Fanuc TP program (LS listing): JOB_VAR_OD_GRIP.LS

/PROG  JOB_VAR_OD_GRIP
/ATTR
OWNER		= MNEDITOR;
COMMENT		= "";
PROG_SIZE	= 93425;
CREATE		= DATE 19-07-31  TIME 17:01:20;
MODIFIED	= DATE 26-06-08  TIME 14:37:38;
FILE_NAME	= JOB_VARI;
VERSION		= 0;
LINE_COUNT = 3201;
MEMORY_SIZE	= 94489;
PROTECT		= READ_WRITE;
TCD:  STACK_SIZE	= 0,
      TASK_PRIORITY	= 50,
      TIME_SLICE	= 0,
      BUSY_LAMP_OFF	= 0,
      ABORT_REQUEST	= 0,
      PAUSE_REQUEST	= 0;
DEFAULT_GROUP	= 1,*,*,*,*;
CONTROL_CODE	= 00000000 00000000;
/APPL

AUTO_SINGULARITY_HEADER;
  ENABLE_SINGULARITY_AVOIDANCE   : TRUE;
/MN
   1:  !R[70] is the item number ;
   2:  !R[71] if using previous data ;
   3:  R[196]=AR[1]    ;
   4:  R[197]=AR[2]    ;
   5:  !------------------------- ;
   6:  !Item Select = 102680550 ;
   7:  SELECT R[70]=550,JMP LBL[550] ;
   8:  !Item Select = 102680552 ;
   9:         =552,JMP LBL[552] ;
  10:  !Item Select = MEC0253 ;
  11:         =253,JMP LBL[253] ;
  12:  !Item Select = 102680551 ;
  13:         =551,JMP LBL[551] ;
  14:  !Item Select = 1090747 ;
  15:         =747,JMP LBL[747] ;
  16:  !Item Select = 102772049 ;
  17:         =2049,JMP LBL[2049] ;
  18:  !Item Select = 102712760 ;
  19:         =2760,JMP LBL[2760] ;
  20:  !Item Select = 102740005 ;
  21:         =4005,JMP LBL[4005] ;
  22:  !Item Select = 103044540 ;
  23:         =4540,JMP LBL[4540] ;
  24:  !Item Select = 102824679 ;
  25:         =4679,JMP LBL[4679] ;
  26:  !Item Select = 103095029 ;
  27:         =5029,JMP LBL[5029] ;
  28:  !Item Select = 1025649 ;
  29:         =5649,JMP LBL[5649] ;
  30:  !Item Select = 103365943 ;
  31:         =5943,JMP LBL[5943] ;
  32:  !Item Select = 102906372 ;
  33:         =6372,JMP LBL[6372] ;
  34:  !Item Select = 102666549 ;
  35:         =6549,JMP LBL[6549] ;
  36:  !Item Select = 1026588 ;
  37:         =6588,JMP LBL[6588] ;
  38:  !Item Select = 1026617 ;
  39:         =6617,JMP LBL[6617] ;
  40:  !Item Select = 102606754 ;
  41:         =6754,JMP LBL[6754] ;
  42:  !Item Select = 102606755 ;
  43:         =6755,JMP LBL[6755] ;
  44:  !Item Select = 102757062 ;
  45:         =7062,JMP LBL[7062] ;
  46:  !Item Select = 102577436 ;
  47:         =7436,JMP LBL[7436] ;
  48:  !Item Select = 1017688 ;
  49:         =7688,JMP LBL[7688] ;
  50:  !Item Select = 207757 ;
  51:         =7757,JMP LBL[7757] ;
  52:  !Item Select = 198034 ;
  53:         =8034,JMP LBL[8034] ;
  54:  !Item Select = 102678902 ;
  55:         =8902,JMP LBL[8902] ;
  56:  !Item Select = 102709487 ;
  57:         =9487,JMP LBL[9487] ;
  58:  !Item Select = 100009654 ;
  59:         =9654,JMP LBL[9654] ;
  60:  !Item Select = 102779700 ;
  61:         =9700,JMP LBL[9700] ;
  62:  !Item Select = 102649814 ;
  63:         =9814,JMP LBL[9814] ;

  64:  !Item Select = 111199990 ;
  65:         =9990,JMP LBL[9990] ;


  66:  !No conditions are met, jump ;
  67:  !to the very end of the program ;
  68:         ELSE,JMP LBL[9999] ;
  69:   ;
  70:  LBL[253] ;
  71:  !--------------------------- ;
  72:  !HANDLE PULL ;
  73:  !Item MEC0253, Rev 01-000 ;
  74:  !Last Modified: 2025-07-25 ;
  75:  !Modified by: AARON ;
  76:  !0.35 IN Height ;
  77:  !0.09 IN ID, 0.25 IN OD ;
  78:  !OD Jaw #1005 ;
  79:  !------------------------- ;
  80:  IF (R[70]=253) THEN ;
  81:   ;
  82:  !Define Parameters for INF/OTF ;
  83:  !R[105]=AR[1]=100, 2By3 Sheet ;
  84:  !R[105]=AR[1]=200, 3By4 Sheet ;
  85:  !R[105]=AR[1]=300, 5By7 Sheet ;
  86:  CALL JOB_VAR_SETUP(200) ;
  87:   ;
  88:  !------------------------- ;
  89:  !Define Parameters for Job ;
  90:  R[1]=0    ;
  91:  R[67]=20    ;
  92:  R[2]=0    ;
  93:  R[3]=1    ;
  94:  R[139]=12    ;
  95:  R[4]=0    ;
  96:  R[85]=64    ;
  97:  R[86]=5    ;
  98:  R[87]=150    ;
  99:  R[95]=100    ;
 100:  R[110]=2026    ;
 101:  !CNC W-AXIS OFFSET ;
 102:  R[111]=((-16.06)) ;
 103:  !X-Compliance Push Bypass ;
 104:  F[6:OFF]=(OFF) ;
 105:  !--------------------------- ;
 106:  !R[100] "GRIPPER_ID" 3 values ;
 107:  !If =100, ID Grippers Installed ;
 108:  !If =200, OD Grippers Installed ;
 109:  !If =300, OD 45 Degree Grippers ;
 110:  R[100]=200    ;
 111:  !--------------------------- ;
 112:   ;
 113:  !If using previous setup data ;
 114:  IF (R[71]=253) THEN ;
 115:   ;
 116:  !--------------------------- ;
 117:  R[190]=20.5    ;
 118:  R[191]=15.798    ;
 119:  R[192]=(-36)    ;
 120:  R[193]=(-440)    ;
 121:  !--------------------------- ;
 122:   ;
 123:   ;
 124:  CALL CREATE_REG(R[190],R[191],R[192],R[193]) ;
 125:   ;
 126:  ENDIF ;
 127:   ;
 128:  !If new loading or offloading pos ;
 129:  !SET R[104] "IMPORT_LOADPOS" ;
 130:  !SET R[104]=1000, Otherwise NO ;
 131:  R[104]=1000    ;
 132:  IF (R[104]=1000) THEN ;
 133:  !R[260]=43, Preload Pos1 ;
 134:  !R[270]=44, Preload PosFinal ;
 135:  !R[300]=53, Offload PosFinal ;
 136:  !PR[43] Pre-Loading Pos1 ;
 137:  CALL CREATE_PR(43,167.761,(-61.029),337.113,(-171.936),88.039,(-174.046)) ;
 138:  !PR[44] Final Loading Position ;
 139:  CALL CREATE_PR(44,168.578,(-60.735),361.702,(-171.929),88.036,(-174.03)) ;
 140:  !PR[53] Pre Unloading Position ;
 141:  CALL CREATE_PR(53,(-127.197),94.302,111.215,163.187,(-88.443),(-162.218)) ;
 142:  !PR[54] Final Unloading Position ;
 143:  CALL CREATE_PR(54,(-125.519),94.106,49.029,163.508,(-88.445),(-162.507)) ;
 144:  ENDIF ;
 145:   ;
 146:  !---------------------------- ;
 147:  !SR[2] = "JOB_VAR_OD_GRIP" ;
 148:  !JOB_VAR_COMMON(R[103])'s value ;
 149:  !---------------------------- ;
 150:  !2By3 SR[2] INF, Max 18(Straight) ;
 151:  !R[103]=200 ;
 152:  !2By3 INF 45 Degree Diagonal Shif ;
 153:  !R[103]=210 ;
 154:  !---------------------------- ;
 155:  !3By4 SR[2] INF, Max 36(Straight) ;
 156:  !R[103]=250 ;
 157:  !3By4 INF 45 Degree Diagonal Shif ;
 158:  !R[103]=260 ;
 159:  !---------------------------- ;
 160:  !R[103] "JOB_PROFILE" Selection ;
 161:  R[103]=250    ;
 162:  CALL JOB_VAR_COMMON(R[103]) ;
 163:   ;
 164:  ENDIF ;
 165:   ;
 166:  JMP LBL[9999] ;
 167:   ;
 168:  !Job MEC0253 Logic Ends ;
 169:  !--------------------------- ;
 170:   ;
 171:  LBL[550] ;
 172:  !--------------------------- ;
 173:  !Thimble Upper ;
 174:  !Item 102680550 , Rev A ;
 175:  !Last Modified: 2024-06-24 ;
 176:  !Modified by: SH ;
 177:  !1.06 IN Height ;
 178:  !3.3 IN ID, 4.49 IN OD ;
 179:  !OD Jaw # 2003 ;
 180:  !--------------------------- ;
 181:  IF (R[70]=550) THEN ;
 182:  !Define Parameters for INF/OTF ;
 183:  !R[105]=AR[1]=100, 2By3 Sheet ;
 184:  !R[105]=AR[1]=200, 3By4 Sheet ;
 185:  !R[105]=AR[1]=300, 5By7 Sheet ;
 186:  CALL JOB_VAR_SETUP(100) ;
 187:   ;
 188:  !--------------------------- ;
 189:  !Define Parameters for Job ;
 190:  R[1]=1    ;
 191:  R[67]=20    ;
 192:  R[2]=0    ;
 193:  R[139]=12    ;
 194:  !R[85] "INF_JAW_OFFSET"(Hgt) ;
 195:  R[85]=92.05    ;
 196:  !R[86] "INF_PICK_OFFSET" 50mm/sec ;
 197:  R[86]=5    ;
 198:  !R[87] "MAIN_LOAD_OFFSET" (PRELOA ;
 199:  R[87]=100    ;
 200:  !R[100] "GRIPPER_ID" 3 values ;
 201:  !If =100, ID Grippers Installed ;
 202:  !If =200, OD Grippers Installed ;
 203:  !If =300, OD 45 Degree Grippers ;
 204:  R[100]=200    ;
 205:  !--------------------------- ;
 206:   ;
 207:  !If using previous setup data ;
 208:  IF (R[71]=550) THEN ;
 209:   ;
 210:  !--------------------------- ;
 211:  !1st: Height of Raw piece ;
 212:  R[190]=32.2    ;
 213:  !2nd: Height of Finish piece ;
 214:  R[191]=27    ;
 215:  !3rd: Infeed Height Offset ;
 216:  R[192]=(-240)    ;
 217:  !4th: Outfeed Height Offset ;
 218:  R[193]=(-285)    ;
 219:  !--------------------------- ;
 220:   ;
 221:  CALL CREATE_REG(R[190],R[191],R[192],R[193]) ;
 222:   ;
 223:  ENDIF ;
 224:   ;
 225:  !If new loading or offloading pos ;
 226:  !SET R[104] "IMPORT_LOADPOS" ;
 227:  !SET R[104]=1000, Otherwise NO ;
 228:  R[104]=1000    ;
 229:  IF (R[104]=1000) THEN ;
 230:  !R[260]=43, Preload Pos1 ;
 231:  !R[270]=44, Preload PosFinal ;
 232:  !R[300]=53, Offload PosFinal ;
 233:  !PR[43] Pre-Loading Pos1 ;
 234:  CALL CREATE_PR(43,167.274,(-59.505),319.711,168.214,88.493,166.138) ;
 235:  !PR[44] Final Loading Position ;
 236:  CALL CREATE_PR(44,167.813,(-59.797),340.237,168.005,88.489,165.921) ;
 237:  !PR[53] Pre Unloading Position ;
 238:  CALL CREATE_PR(53,(-127.387),93.873,91.227,168.522,(-88.33),(-169.447)) ;
 239:  !PR[54] Final Unloading Position ;
 240:  CALL CREATE_PR(54,(-126.716),94.154,67.135,168.491,(-88.33),(-169.421)) ;
 241:  !PR[56] assitant Unloading preses ;
 242:  CALL CREATE_PR(56,(-131.536),105.713,233.177,173.746,(-88.233),(-175.647)) ;
 243:  !PR[57] assitant Unloading preses ;
 244:  CALL CREATE_PR(57,(-133.703),92.431,364.782,167.802,(-88.383),(-166.755)) ;
 245:  !PR[58] assitant Unloading preses ;
 246:  CALL CREATE_PR(58,(-133.703),92.431,364.782,167.804,(-88.383),(-166.755)) ;
 247:  ENDIF ;
 248:   ;
 249:  !---------------------------- ;
 250:  !SR[2] = "JOB_VAR_OD_GRIP" ;
 251:  !JOB_VAR_COMMON(R[103])'s value ;
 252:  !---------------------------- ;
 253:  !2By3 SR[2] INF, Max 18(Straight) ;
 254:  !R[103]=200 ;
 255:  !2By3 INF 45 Degree Diagonal Shif ;
 256:  !R[103]=210 ;
 257:  !---------------------------- ;
 258:  !3By4 SR[2] INF, Max 36(Straight) ;
 259:  !R[103]=250 ;
 260:  !3By4 INF 45 Degree Diagonal Shif ;
 261:  !R[103]=260 ;
 262:  !---------------------------- ;
 263:  !R[103] "JOB_PROFILE" Selection ;
 264:  R[103]=200    ;
 265:  CALL JOB_VAR_COMMON(R[103]) ;
 266:   ;
 267:  ENDIF ;
 268:   ;
 269:  JMP LBL[9999] ;
 270:   ;
 271:  !Job 102680550 Logic Ends ;
 272:  !--------------------------- ;
 273:   ;
 274:  LBL[551] ;
 275:  !--------------------------- ;
 276:  !Thimble Lower ;
 277:  !Item 102680551 , Rev A ;
 278:  !Last Modified: 2026-05-20 ;
 279:  !Modified by: Aaron ;
 280:  !1.38 IN Height ;
 281:  !3.372 IN ID, 4.49 IN OD ;
 282:  !OD Jaw # 2002 ;
 283:  !--------------------------- ;
 284:  IF (R[70]=551) THEN ;
 285:  !Define Parameters for INF/OTF ;
 286:  !R[105]=AR[1]=100, 2By3 Sheet ;
 287:  !R[105]=AR[1]=200, 3By4 Sheet ;
 288:  !R[105]=AR[1]=300, 5By7 Sheet ;
 289:  CALL JOB_VAR_SETUP(100) ;
 290:   ;
 291:  !--------------------------- ;
 292:  !Define Parameters for Job ;
 293:  R[1]=1    ;
 294:  R[67]=20    ;
 295:  R[2]=1    ;
 296:  R[139]=12    ;
 297:  !R[85] "INF_JAW_OFFSET"(Hgt) ;
 298:  R[85]=92.05    ;
 299:  !R[86] "INF_PICK_OFFSET" 50mm/sec ;
 300:  R[86]=10    ;
 301:  !R[87] "MAIN_LOAD_OFFSET" (PRELOA ;
 302:  R[87]=100    ;
 303:  !R[100] "GRIPPER_ID" 3 values ;
 304:  !If =100, ID Grippers Installed ;
 305:  !If =200, OD Grippers Installed ;
 306:  !If =300, OD 45 Degree Grippers ;
 307:  R[100]=200    ;
 308:  !--------------------------- ;
 309:   ;
 310:  !If using previous setup data ;
 311:  IF (R[71]=551) THEN ;
 312:   ;
 313:  !--------------------------- ;
 314:  !1st: Height of Raw piece ;
 315:  R[190]=41.5    ;
 316:  !2nd: Height of Finish piece ;
 317:  R[191]=35.05    ;
 318:  !3rd: Infeed Height Offset ;
 319:  R[192]=(-250)    ;
 320:  !4th: Outfeed Height Offset ;
 321:  R[193]=(-280)    ;
 322:  !--------------------------- ;
 323:   ;
 324:  CALL CREATE_REG(R[190],R[191],R[192],R[193]) ;
 325:   ;
 326:  ENDIF ;
 327:   ;
 328:  !If new loading or offloading pos ;
 329:  !SET R[104] "IMPORT_LOADPOS" ;
 330:  !SET R[104]=1000, Otherwise NO ;
 331:  R[104]=1000    ;
 332:  IF (R[104]=1000) THEN ;
 333:  !R[260]=43, Preload Pos1 ;
 334:  !R[270]=44, Preload PosFinal ;
 335:  !R[300]=53, Offload PosFinal ;
 336:  !PR[43] Pre-Loading Pos1 ;
 337:  CALL CREATE_PR(43,166.588,(-60.843),303.6,142.233,88.871,140.108) ;
 338:  !PR[44] Final Loading Position ;
 339:  CALL CREATE_PR(44,167.032,(-61.379),332.527,142.158,88.868,140.022) ;
 340:  !PR[53] Pre Unloading Position ;
 341:  CALL CREATE_PR(53,(-128.024),95.156,112.32,168.042,(-88.32),(-169.031)) ;
 342:  !PR[54] Final Unloading Position ;
 343:  CALL CREATE_PR(54,(-126.891),94.757,73.15,168.209,(-88.331),(-169.169)) ;
 344:  !PR[56] assitant Unloading preses ;
 345:  CALL CREATE_PR(56,(-131.536),105.713,233.177,173.746,(-88.233),(-175.647)) ;
 346:  !PR[57] assitant Unloading preses ;
 347:  CALL CREATE_PR(57,(-133.703),92.431,364.782,167.802,(-88.383),(-166.755)) ;
 348:  !PR[58] assitant Unloading preses ;
 349:  CALL CREATE_PR(58,(-133.703),92.431,364.782,167.804,(-88.383),(-166.755)) ;
 350:  ENDIF ;
 351:   ;
 352:  !---------------------------- ;
 353:  !SR[2] = "JOB_VAR_OD_GRIP" ;
 354:  !JOB_VAR_COMMON(R[103])'s value ;
 355:  !---------------------------- ;
 356:  !2By3 SR[2] INF, Max 18(Straight) ;
 357:  !R[103]=200 ;
 358:  !2By3 INF 45 Degree Diagonal Shif ;
 359:  !R[103]=210 ;
 360:  !---------------------------- ;
 361:  !3By4 SR[2] INF, Max 36(Straight) ;
 362:  !R[103]=250 ;
 363:  !3By4 INF 45 Degree Diagonal Shif ;
 364:  !R[103]=260 ;
 365:  !---------------------------- ;
 366:  !R[103] "JOB_PROFILE" Selection ;
 367:  R[103]=200    ;
 368:  CALL JOB_VAR_COMMON(R[103]) ;
 369:   ;
 370:  ENDIF ;
 371:   ;
 372:  JMP LBL[9999] ;
 373:   ;
 374:  !Job 102680551 Logic Ends ;
 375:  !--------------------------- ;
 376:   ;
 377:  LBL[552] ;
 378:  !--------------------------- ;
 379:  !COLLAR ;
 380:  !Item 102680552 , Rev A ;
 381:  !Last Modified: 2024-06-25 ;
 382:  !Modified by: TSUU ;
 383:  !1.79 IN Height ;
 384:  !3.110 IN ID, 3.56 IN OD ;
 385:  !OD Jaw # 2002 ;
 386:  !--------------------------- ;
 387:  IF (R[70]=552) THEN ;
 388:  !Define Parameters for INF/OTF ;
 389:  !R[105]=AR[1]=100, 2By3 Sheet ;
 390:  !R[105]=AR[1]=200, 3By4 Sheet ;
 391:  !R[105]=AR[1]=300, 5By7 Sheet ;
 392:  CALL JOB_VAR_SETUP(100) ;
 393:   ;
 394:  !--------------------------- ;
 395:  !Define Parameters for Job ;
 396:  R[1]=1    ;
 397:  R[67]=20    ;
 398:  R[2]=1    ;
 399:  R[139]=12    ;
 400:  !R[85] "INF_JAW_OFFSET"(Hgt) ;
 401:  R[85]=200    ;
 402:  !R[86] "INF_PICK_OFFSET" 50mm/sec ;
 403:  R[86]=15    ;
 404:  !R[87] "MAIN_LOAD_OFFSET" (PRELOA ;
 405:  R[87]=100    ;
 406:  !R[100] "GRIPPER_ID" 3 values ;
 407:  !If =100, ID Grippers Installed ;
 408:  !If =200, OD Grippers Installed ;
 409:  !If =300, OD 45 Degree Grippers ;
 410:  R[100]=200    ;
 411:  !--------------------------- ;
 412:   ;
 413:  !If using previous setup data ;
 414:  IF (R[71]=552) THEN ;
 415:   ;
 416:  !--------------------------- ;
 417:  !1st: Height of Raw piece ;
 418:  R[190]=50.546    ;
 419:  !2nd: Height of Finish piece ;
 420:  R[191]=45.46    ;
 421:  !3rd: Infeed Height Offset ;
 422:  R[192]=(-250)    ;
 423:  !4th: Outfeed Height Offset ;
 424:  R[193]=(-250)    ;
 425:  !--------------------------- ;
 426:   ;
 427:  CALL CREATE_REG(R[190],R[191],R[192],R[193]) ;
 428:   ;
 429:  ENDIF ;
 430:   ;
 431:  !If new loading or offloading pos ;
 432:  !SET R[104] "IMPORT_LOADPOS" ;
 433:  !SET R[104]=1000, Otherwise NO ;
 434:  R[104]=1000    ;
 435:  IF (R[104]=1000) THEN ;
 436:  !R[260]=43, Preload Pos1 ;
 437:  !R[270]=44, Preload PosFinal ;
 438:  !R[300]=53, Offload PosFinal ;
 439:  !PR[43] Pre-Loading Pos1 ;
 440:  CALL CREATE_PR(43,167.759,(-61.04),294.256,160.46,89.14,158.531) ;
 441:  !PR[44] Final Loading Position ;
 442:  CALL CREATE_PR(44,168.25,(-61.377),329.133,160.345,89.147,158.399) ;
 443:  !PR[53] Pre Unloading Position ;
 444:  CALL CREATE_PR(53,(-129.89),93.66,171.06,156.59,(-88.74),(-166.46)) ;
 445:  !PR[54] Final Unloading Position ;
 446:  CALL CREATE_PR(54,(-129),93.98,128.255,156.535,(-88.747),(-166.399)) ;
 447:  !PR[56] assitant Unloading preses ;
 448:  CALL CREATE_PR(56,(-131.536),105.713,233.177,173.746,(-88.233),(-175.647)) ;
 449:  !PR[57] assitant Unloading preses ;
 450:  CALL CREATE_PR(57,(-133.703),92.431,364.782,167.802,(-88.383),(-166.755)) ;
 451:  !PR[58] assitant Unloading preses ;
 452:  CALL CREATE_PR(58,(-133.703),92.431,364.782,167.804,(-88.383),(-166.755)) ;
 453:  ENDIF ;
 454:   ;
 455:  !---------------------------- ;
 456:  !SR[2] = "JOB_VAR_OD_GRIP" ;
 457:  !JOB_VAR_COMMON(R[103])'s value ;
 458:  !---------------------------- ;
 459:  !2By3 SR[2] INF, Max 18(Straight) ;
 460:  !R[103]=200 ;
 461:  !2By3 INF 45 Degree Diagonal Shif ;
 462:  !R[103]=210 ;
 463:  !---------------------------- ;
 464:  !3By4 SR[2] INF, Max 36(Straight) ;
 465:  !R[103]=250 ;
 466:  !3By4 INF 45 Degree Diagonal Shif ;
 467:  !R[103]=260 ;
 468:  !---------------------------- ;
 469:  !R[103] "JOB_PROFILE" Selection ;
 470:  R[103]=200    ;
 471:  CALL JOB_VAR_COMMON(R[103]) ;
 472:   ;
 473:  ENDIF ;
 474:   ;
 475:  JMP LBL[9999] ;
 476:   ;
 477:  !Job 102680552 Logic Ends ;
 478:  !--------------------------- ;
 479:   ;
 480:  LBL[747] ;
 481:  !--------------------------- ;
 482:  !PORT-GROVE VENT, JUICEBOX ;
 483:  !Item 1090747, Rev A ;
 484:  !Last Modified: 2025-03-22 ;
 485:  !Modified by: ZAMAN ;
 486:  !0.622 IN Height ;
 487:  !1.202 IN ID, 3.00 IN OD ;
 488:  !OD Jaw #2009 ;
 489:  !------------------------- ;
 490:  IF (R[70]=747) THEN ;
 491:   ;
 492:  !Define Parameters for INF/OTF ;
 493:  !R[105]=AR[1]=100, 2By3 Sheet ;
 494:  !R[105]=AR[1]=200, 3By4 Sheet ;
 495:  !R[105]=AR[1]=300, 5By7 Sheet ;
 496:  CALL JOB_VAR_SETUP(200) ;
 497:   ;
 498:  !------------------------- ;
 499:  !Define Parameters for Job ;
 500:  R[1]=1    ;
 501:  R[67]=20    ;
 502:  R[2]=0    ;
 503:  R[139]=12    ;
 504:  R[3]=0    ;
 505:  R[4]=0    ;
 506:  R[85]=64    ;
 507:  R[86]=5    ;
 508:  R[87]=150    ;
 509:  R[95]=100    ;
 510:  R[110]=2026    ;
 511:  !CNC W-AXIS OFFSET ;
 512:  R[111]=((-16.06)) ;
 513:  !X-Compliance Push Bypass ;
 514:  F[6:OFF]=(OFF) ;
 515:  !--------------------------- ;
 516:  !R[100] "GRIPPER_ID" 3 values ;
 517:  !If =100, ID Grippers Installed ;
 518:  !If =200, OD Grippers Installed ;
 519:  !If =300, OD 45 Degree Grippers ;
 520:  R[100]=200    ;
 521:  !--------------------------- ;
 522:   ;
 523:  !If using previous setup data ;
 524:  IF (R[71]=747) THEN ;
 525:   ;
 526:  !--------------------------- ;
 527:  R[190]=20.5    ;
 528:  R[191]=15.798    ;
 529:  R[192]=(-36)    ;
 530:  R[193]=(-498)    ;
 531:  !--------------------------- ;
 532:   ;
 533:   ;
 534:  CALL CREATE_REG(R[190],R[191],R[192],R[193]) ;
 535:   ;
 536:  ENDIF ;
 537:   ;
 538:  !If new loading or offloading pos ;
 539:  !SET R[104] "IMPORT_LOADPOS" ;
 540:  !SET R[104]=1000, Otherwise NO ;
 541:  R[104]=1000    ;
 542:  IF (R[104]=1000) THEN ;
 543:  !R[260]=43, Preload Pos1 ;
 544:  !R[270]=44, Preload PosFinal ;
 545:  !R[300]=53, Offload PosFinal ;
 546:  !PR[43] Pre-Loading Pos1 ;
 547:  CALL CREATE_PR(43,167.761,(-61.029),337.113,(-171.936),88.039,(-174.046)) ;
 548:  !PR[44] Final Loading Position ;
 549:  CALL CREATE_PR(44,168.578,(-60.735),361.702,(-171.929),88.036,(-174.03)) ;
 550:  !PR[53] Pre Unloading Position ;
 551:  CALL CREATE_PR(53,(-127.197),94.302,111.215,163.187,(-88.443),(-162.218)) ;
 552:  !PR[54] Final Unloading Position ;
 553:  CALL CREATE_PR(54,(-125.536),94.555,48.721,163.38,(-88.442),(-162.397)) ;
 554:  ENDIF ;
 555:   ;
 556:  !---------------------------- ;
 557:  !SR[2] = "JOB_VAR_OD_GRIP" ;
 558:  !JOB_VAR_COMMON(R[103])'s value ;
 559:  !---------------------------- ;
 560:  !2By3 SR[2] INF, Max 18(Straight) ;
 561:  !R[103]=200 ;
 562:  !2By3 INF 45 Degree Diagonal Shif ;
 563:  !R[103]=210 ;
 564:  !---------------------------- ;
 565:  !3By4 SR[2] INF, Max 36(Straight) ;
 566:  !R[103]=250 ;
 567:  !3By4 INF 45 Degree Diagonal Shif ;
 568:  !R[103]=260 ;
 569:  !---------------------------- ;
 570:  !R[103] "JOB_PROFILE" Selection ;
 571:  R[103]=250    ;
 572:  CALL JOB_VAR_COMMON(R[103]) ;
 573:   ;
 574:  ENDIF ;
 575:   ;
 576:  JMP LBL[9999] ;
 577:   ;
 578:  !Job 1090747 Logic Ends ;
 579:  !--------------------------- ;
 580:   ;
 581:  LBL[2049] ;
 582:  !--------------------------- ;
 583:  !Mandrel ;
 584:  !Item 102772049 , Rev A ;
 585:  !Last Modified: 2022-04-09 ;
 586:  !Modified by: Tsuu ;
 587:  !17.24 IN Height ;
 588:  !3.22 IN ID, 1.00 IN OD ;
 589:  !OD Jaw #2006 ;
 590:  !--------------------------- ;
 591:  IF (R[70]=2049) THEN ;
 592:  !Define Parameters for INF/OTF ;
 593:  !R[105]=AR[1]=100, 2By3 Sheet ;
 594:  !R[105]=AR[1]=200, 3By4 Sheet ;
 595:  !R[105]=AR[1]=210, 3By4 Sheet Man ;
 596:  !R[105]=AR[1]=300, 5By7 Sheet ;
 597:  CALL JOB_VAR_SETUP(210) ;
 598:   ;
 599:  !--------------------------- ;
 600:  !Define Parameters for Job ;
 601:  !R[85] "INF_JAW_OFFSET"(Hgt) ;
 602:  R[85]=55    ;
 603:  !R[86] "INF_PICK_OFFSET" 50mm/sec ;
 604:  R[86]=40    ;
 605:  !R[87] "MAIN_LOAD_OFFSET" (PRELOA ;
 606:  R[87]=0    ;
 607:  !R[100] "GRIPPER_ID" 3 values ;
 608:  !If =100, ID Grippers Installed ;
 609:  !If =200, OD Grippers Installed ;
 610:  !If =300, OD 45 Degree Grippers ;
 611:  R[100]=200    ;
 612:  !--------------------------- ;
 613:   ;
 614:  !If using previous setup data ;
 615:  IF (R[71]=2049) THEN ;
 616:   ;
 617:  !--------------------------- ;
 618:  !1st: Height of Raw piece ;
 619:  R[190]=450    ;
 620:  !2nd: Height of Finish piece ;
 621:  R[191]=437.896    ;
 622:  !3rd: Infeed Height Offset ;
 623:  R[192]=(-500)    ;
 624:  !4th: Outfeed Height Offset ;
 625:  R[193]=(-180)    ;
 626:  !--------------------------- ;
 627:   ;
 628:  CALL CREATE_REG(R[190],R[191],R[192],R[193]) ;
 629:   ;
 630:  ENDIF ;
 631:   ;
 632:  !If new loading or offloading pos ;
 633:  !SET R[104] "IMPORT_LOADPOS" ;
 634:  !SET R[104]=1000, Otherwise NO ;
 635:  R[104]=1000    ;
 636:  IF (R[104]=1000) THEN ;
 637:  !R[260]=43, Preload Pos1 ;
 638:  !R[270]=44, Preload PosFinal ;
 639:  !R[300]=53, Offload PosFinal ;
 640:  !PR[43] Pre-Loading Pos1 ;
 641:  CALL CREATE_PR(43,160.063,(-59.564),(-124.262),136.643,88.833,134.535) ;
 642:  !PR[44] Final Loading Position ;
 643:  CALL CREATE_PR(44,163.064,(-60.998),20.902,136.802,88.823,134.669) ;
 644:  !PR[53] Pre Unloading Position ;
 645:  CALL CREATE_PR(53,(-129.19),94.821,118.922,173.603,(-88.242),(-175.552)) ;
 646:  !PR[54] Final Unloading Position ;
 647:  CALL CREATE_PR(54,(-127.505),95.049,62.976,173.55,(-88.244),(-175.503)) ;
 648:  !PR[56] assitant Unloading preses ;
 649:  CALL CREATE_PR(56,(-131.298),94.552,188.064,173.651,(-88.242),(-175.595)) ;
 650:  !PR[57] assitant Unloading preses ;
 651:  CALL CREATE_PR(57,(-133.938),94.235,274.821,173.733,(-88.241),(-175.673)) ;
 652:  !PR[58] assitant Unloading preses ;
 653:  CALL CREATE_PR(58,(-136.182),93.951,348.894,173.814,(-88.239),(-175.748)) ;
 654:  !PR[59] assitant Unloading preses ;
 655:  CALL CREATE_PR(59,82.383,234.843,398.401,(-92.773),(-50.7),90.238) ;
 656:  ENDIF ;
 657:   ;
 658:  !---------------------------- ;
 659:  !SR[2] = "JOB_VAR_OD_GRIP" ;
 660:  !JOB_VAR_COMMON(R[103])'s value ;
 661:  !---------------------------- ;
 662:  !2By3 SR[2] INF, Max 18(Straight) ;
 663:  !R[103]=200 ;
 664:  !2By3 INF 45 Degree Diagonal Shif ;
 665:  !R[103]=210 ;
 666:  !---------------------------- ;
 667:  !3By4 SR[2] INF, Max 36(Straight) ;
 668:  !R[103]=250 ;
 669:  !3By4 INF Mandrel, 2 Trays ;
 670:  !R[103]=260 ;
 671:  !---------------------------- ;
 672:  !R[103] "JOB_PROFILE" Selection ;
 673:  R[103]=260    ;
 674:  CALL JOB_VAR_COMMON(R[103]) ;
 675:   ;
 676:  ENDIF ;
 677:   ;
 678:  JMP LBL[9999] ;
 679:   ;
 680:  !Job 102772049 Logic Ends ;
 681:  !--------------------------- ;
 682:   ;
 683:  LBL[2760] ;
 684:  !--------------------------- ;
 685:  !Mandrel ;
 686:  !Item 102712760 , Rev B ;
 687:  !Last Modified: 2022-04-20 ;
 688:  !Modified by: Tsuu ;
 689:  !13.64 IN Height ;
 690:  !1.3 IN ID, 3.08 IN OD ;
 691:  !OD Jaw # 2006 ;
 692:  !--------------------------- ;
 693:  IF (R[70]=2760) THEN ;
 694:  !Define Parameters for INF/OTF ;
 695:  !R[105]=AR[1]=100, 2By3 Sheet ;
 696:  !R[105]=AR[1]=200, 3By4 Sheet ;
 697:  !R[105]=AR[1]=210, 3By4 Sheet Man ;
 698:  !R[105]=AR[1]=300, 5By7 Sheet ;
 699:  CALL JOB_VAR_SETUP(210) ;
 700:   ;
 701:  !--------------------------- ;
 702:  !Define Parameters for Job ;
 703:  !R[85] "INF_JAW_OFFSET"(Hgt) ;
 704:  R[85]=55    ;
 705:  !R[86] "INF_PICK_OFFSET" 50mm/sec ;
 706:  R[86]=40    ;
 707:  !R[87] "MAIN_LOAD_OFFSET" (PRELOA ;
 708:  R[87]=0    ;
 709:  !R[100] "GRIPPER_ID" 3 values ;
 710:  !If =100, ID Grippers Installed ;
 711:  !If =200, OD Grippers Installed ;
 712:  !If =300, OD 45 Degree Grippers ;
 713:  R[100]=200    ;
 714:  !--------------------------- ;
 715:   ;
 716:  !If using previous setup data ;
 717:  IF (R[71]=2760) THEN ;
 718:   ;
 719:  !--------------------------- ;
 720:  !1st: Height of Raw piece ;
 721:  R[190]=350    ;
 722:  !2nd: Height of Finish piece ;
 723:  R[191]=346.454    ;
 724:  !3rd: Infeed Height Offset ;
 725:  R[192]=(-487)    ;
 726:  !4th: Outfeed Height Offset ;
 727:  R[193]=(-279)    ;
 728:  !--------------------------- ;
 729:   ;
 730:  CALL CREATE_REG(R[190],R[191],R[192],R[193]) ;
 731:   ;
 732:  ENDIF ;
 733:   ;
 734:  !If new loading or offloading pos ;
 735:  !SET R[104] "IMPORT_LOADPOS" ;
 736:  !SET R[104]=1000, Otherwise NO ;
 737:  R[104]=1000    ;
 738:  IF (R[104]=1000) THEN ;
 739:  !R[260]=43, Preload Pos1 ;
 740:  !R[270]=44, Preload PosFinal ;
 741:  !R[300]=53, Offload PosFinal ;
 742:  !PR[43] Pre-Loading Pos1 ;
 743:  CALL CREATE_PR(43,161.794,(-59.04),(-31.912),125.009,88.976,123.003) ;
 744:  !PR[44] Final Loading Position ;
 745:  CALL CREATE_PR(44,164.987,(-60.778),114.073,125.217,88.987,123.177) ;
 746:  !PR[53] Pre Unloading Position ;
 747:  CALL CREATE_PR(53,(-129.19),94.821,118.922,173.603,(-88.242),(-175.552)) ;
 748:  !PR[54] Final Unloading Position ;
 749:  CALL CREATE_PR(54,(-126.806),95.411,40.963,173.785,(-88.244),(-175.725)) ;
 750:  !PR[56] assitant Unloading preses ;
 751:  CALL CREATE_PR(56,(-131.298),94.552,188.064,173.651,(-88.242),(-175.595)) ;
 752:  !PR[57] assitant Unloading preses ;
 753:  CALL CREATE_PR(57,(-133.938),94.235,274.821,173.733,(-88.241),(-175.673)) ;
 754:  !PR[58] assitant Unloading preses ;
 755:  CALL CREATE_PR(58,(-136.182),93.951,348.894,173.814,(-88.239),(-175.748)) ;
 756:  !PR[59] assitant Unloading preses ;
 757:  CALL CREATE_PR(59,82.383,234.843,398.401,(-92.773),0,90.238) ;
 758:  ENDIF ;
 759:   ;
 760:  !---------------------------- ;
 761:  !SR[2] = "JOB_VAR_OD_GRIP" ;
 762:  !JOB_VAR_COMMON(R[103])'s value ;
 763:  !---------------------------- ;
 764:  !2By3 SR[2] INF, Max 18(Straight) ;
 765:  !R[103]=200 ;
 766:  !2By3 INF 45 Degree Diagonal Shif ;
 767:  !R[103]=210 ;
 768:  !---------------------------- ;
 769:  !3By4 SR[2] INF, Max 36(Straight) ;
 770:  !R[103]=250 ;
 771:  !3By4 INF Mandrel, 2 Trays ;
 772:  !R[103]=260 ;
 773:  !---------------------------- ;
 774:  !R[103] "JOB_PROFILE" Selection ;
 775:  R[103]=260    ;
 776:  CALL JOB_VAR_COMMON(R[103]) ;
 777:   ;
 778:  ENDIF ;
 779:   ;
 780:  JMP LBL[9999] ;
 781:   ;
 782:  !Job 102712760 Logic Ends ;
 783:  !--------------------------- ;
 784:   ;
 785:  LBL[4005] ;
 786:  !--------------------------- ;
 787:  !Mandrel ;
 788:  !Item 102740005 , Rev xxx ;
 789:  !Last Modified: 2022-04-22 ;
 790:  !Modified by: Tsuu ;
 791:  !16.25 IN Height ;
 792:  !1.3 IN ID, 3.22 IN OD ;
 793:  !ID Jaw # 2006 ;
 794:  !--------------------------- ;
 795:  IF (R[70]=4005) THEN ;
 796:  !Define Parameters for INF/OTF ;
 797:  !R[105]=AR[1]=100, 2By3 Sheet ;
 798:  !R[105]=AR[1]=200, 3By4 Sheet ;
 799:  !R[105]=AR[1]=210, 3By4 Sheet Man ;
 800:  !R[105]=AR[1]=300, 5By7 Sheet ;
 801:  CALL JOB_VAR_SETUP(210) ;
 802:   ;
 803:  !--------------------------- ;
 804:  !Define Parameters for Job ;
 805:  !R[85] "INF_JAW_OFFSET"(Hgt) ;
 806:  R[85]=55    ;
 807:  !R[86] "INF_PICK_OFFSET" 50mm/sec ;
 808:  R[86]=20    ;
 809:  !R[87] "MAIN_LOAD_OFFSET" (PRELOA ;
 810:  R[87]=0    ;
 811:  !R[100] "GRIPPER_ID" 3 values ;
 812:  !If =100, ID Grippers Installed ;
 813:  !If =200, OD Grippers Installed ;
 814:  !If =300, OD 45 Degree Grippers ;
 815:  R[100]=200    ;
 816:  !--------------------------- ;
 817:   ;
 818:  !If using previous setup data ;
 819:  IF (R[71]=4005) THEN ;
 820:   ;
 821:  !--------------------------- ;
 822:  !1st: Height of Raw piece ;
 823:  R[190]=416    ;
 824:  !2nd: Height of Finish piece ;
 825:  R[191]=412.75    ;
 826:  !3rd: Infeed Height Offset ;
 827:  R[192]=(-488)    ;
 828:  !4th: Outfeed Height Offset ;
 829:  R[193]=(-235)    ;
 830:  !--------------------------- ;
 831:   ;
 832:  CALL CREATE_REG(R[190],R[191],R[192],R[193]) ;
 833:   ;
 834:  ENDIF ;
 835:   ;
 836:  !If new loading or offloading pos ;
 837:  !SET R[104] "IMPORT_LOADPOS" ;
 838:  !SET R[104]=1000, Otherwise NO ;
 839:  R[104]=1000    ;
 840:  IF (R[104]=1000) THEN ;
 841:  !R[260]=43, Preload Pos1 ;
 842:  !R[270]=44, Preload PosFinal ;
 843:  !R[300]=53, Offload PosFinal ;
 844:  !PR[43] Pre-Loading Pos1 ;
 845:  CALL CREATE_PR(43,160.851,(-59.576),(-94.146),125.352,88.898,123.291) ;
 846:  !PR[44] Final Loading Position ;
 847:  CALL CREATE_PR(44,163.299,(-60.879),48.016,137.171,88.811,135.063) ;
 848:  !PR[53] Pre Unloading Position ;
 849:  CALL CREATE_PR(53,(-131.61),94.273,206.06,170.153,(-88.46),(-172.016)) ;
 850:  !PR[54] Final Unloading Position ;
 851:  CALL CREATE_PR(54,(-129.962),94.592,143.929,170.147,(-88.459),(-172.011)) ;
 852:  !PR[56] assitant Unloading preses ;
 853:  CALL CREATE_PR(56,(-132.37),94.143,228.533,172.093,(-88.333),(-173.994)) ;
 854:  !PR[57] assitant Unloading preses ;
 855:  CALL CREATE_PR(57,(-134.362),93.83,298.01,172.16,(-88.331),(-174.054)) ;
 856:  !PR[58] assitant Unloading preses ;
 857:  CALL CREATE_PR(58,(-136.182),93.951,348.894,173.814,(-88.239),(-175.748)) ;
 858:  !PR[59] assitant Unloading preses ;
 859:  CALL CREATE_PR(59,82.373,234.687,398.527,(-91.753),0,88.068) ;
 860:  ENDIF ;
 861:   ;
 862:  !---------------------------- ;
 863:  !SR[2] = "JOB_VAR_OD_GRIP" ;
 864:  !JOB_VAR_COMMON(R[103])'s value ;
 865:  !---------------------------- ;
 866:  !2By3 SR[2] INF, Max 18(Straight) ;
 867:  !R[103]=200 ;
 868:  !2By3 INF 45 Degree Diagonal Shif ;
 869:  !R[103]=210 ;
 870:  !---------------------------- ;
 871:  !3By4 SR[2] INF, Max 36(Straight) ;
 872:  !R[103]=250 ;
 873:  !3By4 INF Mandrel, 2 Trays ;
 874:  !R[103]=260 ;
 875:  !---------------------------- ;
 876:  !R[103] "JOB_PROFILE" Selection ;
 877:  R[103]=260    ;
 878:  CALL JOB_VAR_COMMON(R[103]) ;
 879:   ;
 880:  ENDIF ;
 881:   ;
 882:  JMP LBL[9999] ;
 883:   ;
 884:  !Job 102740005 Logic Ends ;
 885:  !--------------------------- ;
 886:   ;
 887:  LBL[4540] ;
 888:  !--------------------------- ;
 889:  !Wedge ;
 890:  !Item 103044540 , Rev B ;
 891:  !Last Modified: 2023-02-22 ;
 892:  !Modified by: Tsuu ;
 893:  !3.60 IN Height ;
 894:  !1.50 IN ID, 4.30 IN OD ;
 895:  !OD Jaw # 2002 ;
 896:  !--------------------------- ;
 897:  IF (R[70]=4540) THEN ;
 898:  !Define Parameters for INF/OTF ;
 899:  !R[105]=AR[1]=100, 2By3 Sheet ;
 900:  !R[105]=AR[1]=200, 3By4 Sheet ;
 901:  !R[105]=AR[1]=300, 5By7 Sheet ;
 902:  CALL JOB_VAR_SETUP(100) ;
 903:   ;
 904:  !--------------------------- ;
 905:  !Define Parameters for Job ;
 906:  !R[85] "INF_JAW_OFFSET"(Hgt) ;
 907:  R[85]=90    ;
 908:  !R[86] "INF_PICK_OFFSET" 50mm/sec ;
 909:  R[86]=10    ;
 910:  !R[87] "MAIN_LOAD_OFFSET" (PRELOA ;
 911:  R[87]=100    ;
 912:  !R[100] "GRIPPER_ID" 3 values ;
 913:  !If =100, ID Grippers Installed ;
 914:  !If =200, OD Grippers Installed ;
 915:  !If =300, OD 45 Degree Grippers ;
 916:  R[100]=200    ;
 917:  !--------------------------- ;
 918:   ;
 919:  !If using previous setup data ;
 920:  IF (R[71]=4540) THEN ;
 921:   ;
 922:  !--------------------------- ;
 923:  !1st: Height of Raw piece ;
 924:  R[190]=93.98    ;
 925:  !2nd: Height of Finish piece ;
 926:  R[191]=91.44    ;
 927:  !3rd: Infeed Height Offset ;
 928:  R[192]=(-280)    ;
 929:  !4th: Outfeed Height Offset ;
 930:  R[193]=(-270)    ;
 931:  !--------------------------- ;
 932:   ;
 933:  CALL CREATE_REG(R[190],R[191],R[192],R[193]) ;
 934:   ;
 935:  ENDIF ;
 936:   ;
 937:  !If new loading or offloading pos ;
 938:  !SET R[104] "IMPORT_LOADPOS" ;
 939:  !SET R[104]=1000, Otherwise NO ;
 940:  R[104]=1000    ;
 941:  IF (R[104]=1000) THEN ;
 942:  !R[260]=43, Preload Pos1 ;
 943:  !R[270]=44, Preload PosFinal ;
 944:  !R[300]=53, Offload PosFinal ;
 945:  !PR[43] Pre-Loading Pos1 ;
 946:  CALL CREATE_PR(43,168.391,(-60.54),311.539,142.286,89.156,140.304) ;
 947:  !PR[44] Final Loading Position ;
 948:  CALL CREATE_PR(44,168.694,(-60.882),337.079,142.296,89.156,140.31) ;
 949:  !PR[53] Pre Unloading Position ;
 950:  CALL CREATE_PR(53,(-125.075),94.769,57.235,168.207,(-88.383),(-167.145)) ;
 951:  !PR[54] Final Unloading Position ;
 952:  CALL CREATE_PR(54,(-122.937),95.366,(-21.188),168.195,(-88.383),(-167.136)) ;
 953:  !PR[56] assitant Unloading preses ;
 954:  CALL CREATE_PR(56,(-131.536),105.713,233.177,173.746,(-88.233),(-175.647)) ;
 955:  !PR[57] assitant Unloading preses ;
 956:  CALL CREATE_PR(57,(-133.703),92.431,364.782,167.802,(-88.383),(-166.755)) ;
 957:  !PR[58] assitant Unloading preses ;
 958:  CALL CREATE_PR(58,(-133.703),92.431,364.782,167.804,(-88.383),(-166.755)) ;
 959:  ENDIF ;
 960:   ;
 961:  !---------------------------- ;
 962:  !SR[2] = "JOB_VAR_OD_GRIP" ;
 963:  !JOB_VAR_COMMON(R[103])'s value ;
 964:  !---------------------------- ;
 965:  !2By3 SR[2] INF, Max 18(Straight) ;
 966:  !R[103]=200 ;
 967:  !2By3 INF 45 Degree Diagonal Shif ;
 968:  !R[103]=210 ;
 969:  !---------------------------- ;
 970:  !3By4 SR[2] INF, Max 36(Straight) ;
 971:  !R[103]=250 ;
 972:  !3By4 INF 45 Degree Diagonal Shif ;
 973:  !R[103]=260 ;
 974:  !---------------------------- ;
 975:  !R[103] "JOB_PROFILE" Selection ;
 976:  R[103]=200    ;
 977:  CALL JOB_VAR_COMMON(R[103]) ;
 978:   ;
 979:  ENDIF ;
 980:   ;
 981:  JMP LBL[9999] ;
 982:   ;
 983:  !Job 103044540 Logic Ends ;
 984:  !--------------------------- ;
 985:   ;
 986:  LBL[4679] ;
 987:  !--------------------------- ;
 988:  !Jumper Coupling ;
 989:  !Item 102824679 , Rev xxx ;
 990:  !Last Modified: 2021-02-23 ;
 991:  !Modified by: Tsuu ;
 992:  !14.0 IN Height ;
 993:  !0.786 IN ID, 1.25 IN OD ;
 994:  !OD Jaw #2011 ;
 995:  !--------------------------- ;
 996:  IF (R[70]=4679) THEN ;
 997:  !Define Parameters for INF/OTF ;
 998:  !R[105]=AR[1]=100, 2By3 Sheet ;
 999:  !R[105]=AR[1]=200, 3By4 Sheet ;
1000:  !R[105]=AR[1]=300, 5By7 Sheet ;
1001:  CALL JOB_VAR_SETUP(300) ;
1002:   ;
1003:  !--------------------------- ;
1004:  !Define Parameters for Job ;
1005:  !R[85] "INF_JAW_OFFSET"(Hgt) ;
1006:  R[85]=97    ;
1007:  !R[86] "INF_PICK_OFFSET" 50mm/sec ;
1008:  R[86]=0    ;
1009:  !R[87] "MAIN_LOAD_OFFSET" (PRELOA ;
1010:  R[87]=50    ;
1011:  !R[100] "GRIPPER_ID" 3 values ;
1012:  !If =100, ID Grippers Installed ;
1013:  !If =200, OD Grippers Installed ;
1014:  !If =300, OD 45 Degree Grippers ;
1015:  R[100]=200    ;
1016:  !--------------------------- ;
1017:   ;
1018:  !If using previous setup data ;
1019:  IF (R[71]=4679) THEN ;
1020:   ;
1021:  !--------------------------- ;
1022:  !1st: Height of Raw piece ;
1023:  R[190]=355.6    ;
1024:  !2nd: Height of Finish piece ;
1025:  R[191]=355.6    ;
1026:  !3rd: Infeed Height Offset ;
1027:  R[192]=(-243)    ;
1028:  !4th: Outfeed Height Offset ;
1029:  R[193]=(-135)    ;
1030:  !--------------------------- ;
1031:   ;
1032:  CALL CREATE_REG(R[190],R[191],R[192],R[193]) ;
1033:   ;
1034:  ENDIF ;
1035:   ;
1036:  !If new loading or offloading pos ;
1037:  !SET R[104] "IMPORT_LOADPOS" ;
1038:  !SET R[104]=1000, Otherwise NO ;
1039:  R[104]=1000    ;
1040:  IF (R[104]=1000) THEN ;
1041:  !R[260]=43, Preload Pos1 ;
1042:  !R[270]=44, Preload PosFinal ;
1043:  !R[300]=53, Offload PosFinal ;
1044:  !PR[43] Pre-Loading Pos1 ;
1045:  CALL CREATE_PR(43,165.356,(-72.417),(-26.998),172.533,89.126,170.544) ;
1046:  !PR[44] Final Loading Position ;
1047:  CALL CREATE_PR(44,171.778,(-71.125),265.889,159.688,89.07,157.667) ;
1048:  !PR[53] Pre Unloading Position ;
1049:  CALL CREATE_PR(53,(-128.649),108.323,115.549,173.483,(-88.242),(-175.439)) ;
1050:  !PR[54] Final Unloading Position ;
1051:  CALL CREATE_PR(54,(-126.802),108.62,54.262,173.459,(-88.244),(-175.422)) ;
1052:  !PR[56] assitant Unloading preses ;
1053:  CALL CREATE_PR(56,(-131.536),105.713,233.177,173.746,(-88.233),(-175.647)) ;
1054:  !PR[57] assitant Unloading preses ;
1055:  CALL CREATE_PR(57,(-131.536),105.713,233.177,173.746,(-88.233),(-175.647)) ;
1056:  !PR[58] assitant Unloading preses ;
1057:  CALL CREATE_PR(58,(-131.536),105.713,233.177,173.746,(-88.233),(-175.647)) ;
1058:  ENDIF ;
1059:   ;
1060:  !---------------------------- ;
1061:  !SR[2] = "JOB_VAR_OD_GRIP" ;
1062:  !JOB_VAR_COMMON(R[103])'s value ;
1063:  !---------------------------- ;
1064:  !2By3 SR[2] INF, Max 18(Straight) ;
1065:  !R[103]=200 ;
1066:  !2By3 INF 45 Degree Diagonal Shif ;
1067:  !R[103]=210 ;
1068:  !---------------------------- ;
1069:  !3By4 SR[2] INF, Max 36(Straight) ;
1070:  !R[103]=250 ;
1071:  !3By4 INF 45 Degree Diagonal Shif ;
1072:  !R[103]=260 ;
1073:  !---------------------------- ;
1074:  !R[103] "JOB_PROFILE" Selection ;
1075:  R[103]=250    ;
1076:  CALL JOB_VAR_COMMON(R[103]) ;
1077:   ;
1078:  ENDIF ;
1079:   ;
1080:  JMP LBL[9999] ;
1081:   ;
1082:  !Job 102824679 Logic Ends ;
1083:  !--------------------------- ;
1084:   ;
1085:  LBL[5029] ;
1086:  !--------------------------- ;
1087:  !Slip,4X SN235 Buttons ;
1088:  !Item 103095029 , Rev C ;
1089:  !Last Modified: 2023-09-28 ;
1090:  !Modified by: Tsuu, sH ;
1091:  !2.63 IN Height ;
1092:  !2.6 IN ID, 3.36 IN OD ;
1093:  !OD Jaw # 2010 ;
1094:  !--------------------------- ;
1095:  IF (R[70]=5029) THEN ;
1096:  !Define Parameters for INF/OTF ;
1097:  !R[105]=AR[1]=100, 2By3 Sheet ;
1098:  !R[105]=AR[1]=200, 3By4 Sheet ;
1099:  !R[105]=AR[1]=300, 5By7 Sheet ;
1100:  CALL JOB_VAR_SETUP(200) ;
1101:   ;
1102:  !--------------------------- ;
1103:  !Define Parameters for Job ;
1104:  !R[85] "INF_JAW_OFFSET"(Hgt) ;
1105:  R[85]=42.75    ;
1106:  !R[86] "INF_PICK_OFFSET" 50mm/sec ;
1107:  R[86]=15    ;
1108:  !R[87] "MAIN_LOAD_OFFSET" (PRELOA ;
1109:  R[87]=100    ;
1110:  !R[100] "GRIPPER_ID" 3 values ;
1111:  !If =100, ID Grippers Installed ;
1112:  !If =200, OD Grippers Installed ;
1113:  !If =300, OD 45 Degree Grippers ;
1114:  R[100]=200    ;
1115:  !--------------------------- ;
1116:   ;
1117:  !If using previous setup data ;
1118:  IF (R[71]=5029) THEN ;
1119:   ;
1120:  !--------------------------- ;
1121:  !1st: Height of Raw piece ;
1122:  R[190]=70    ;
1123:  !2nd: Height of Finish piece ;
1124:  R[191]=66.802    ;
1125:  !3rd: Infeed Height Offset ;
1126:  R[192]=(-70)    ;
1127:  !4th: Outfeed Height Offset ;
1128:  R[193]=(-455)    ;
1129:  !--------------------------- ;
1130:   ;
1131:  CALL CREATE_REG(R[190],R[191],R[192],R[193]) ;
1132:   ;
1133:  ENDIF ;
1134:   ;
1135:  !If new loading or offloading pos ;
1136:  !SET R[104] "IMPORT_LOADPOS" ;
1137:  !SET R[104]=1000, Otherwise NO ;
1138:  R[104]=1000    ;
1139:  IF (R[104]=1000) THEN ;
1140:  !R[260]=43, Preload Pos1 ;
1141:  !R[270]=44, Preload PosFinal ;
1142:  !R[300]=53, Offload PosFinal ;
1143:  !PR[43] Pre-Loading Pos1 ;
1144:  CALL CREATE_PR(43,167.407,(-61.235),358.579,146.046,89.112,144.041) ;
1145:  !PR[44] Final Loading Position ;
1146:  CALL CREATE_PR(44,167.615,(-61.467),374.198,146.08,89.112,144.08) ;
1147:  !PR[53] Pre Unloading Position ;
1148:  CALL CREATE_PR(53,(-127.197),94.302,111.215,163.187,(-88.443),(-162.218)) ;
1149:  !PR[54] Final Unloading Position ;
1150:  CALL CREATE_PR(54,(-126.244),94.738,73.363,163.118,(-88.444),(-162.154)) ;
1151:  ENDIF ;
1152:   ;
1153:  !---------------------------- ;
1154:  !SR[2] = "JOB_VAR_OD_GRIP" ;
1155:  !JOB_VAR_COMMON(R[103])'s value ;
1156:  !---------------------------- ;
1157:  !2By3 SR[2] INF, Max 18(Straight) ;
1158:  !R[103]=200 ;
1159:  !2By3 INF 45 Degree Diagonal Shif ;
1160:  !R[103]=210 ;
1161:  !---------------------------- ;
1162:  !3By4 SR[2] INF, Max 36(Straight) ;
1163:  !R[103]=250 ;
1164:  !3By4 INF 45 Degree Diagonal Shif ;
1165:  !R[103]=260 ;
1166:  !---------------------------- ;
1167:  !R[103] "JOB_PROFILE" Selection ;
1168:  R[103]=250    ;
1169:  CALL JOB_VAR_COMMON(R[103]) ;
1170:   ;
1171:  ENDIF ;
1172:   ;
1173:  JMP LBL[9999] ;
1174:   ;
1175:  !Job 103095029 Logic Ends ;
1176:  !--------------------------- ;
1177:   ;
1178:  LBL[5649] ;
1179:  !------------------------- ;
1180:  !PISTON ;
1181:  !Item 1025649 ,Rev A ;
1182:  !Last Modified: 2023-12-01 ;
1183:  !Modified by: Tsuu ;
1184:  !0.540 IN Hgt ;
1185:  !0.5 IN ID, 0.987 IN OD ;
1186:  !OD Jaw #2011 ;
1187:  !--------------------------- ;
1188:  IF (R[70]=5649) THEN ;
1189:  !Define Parameters for INF/OTF ;
1190:  !R[105]=AR[1]=100, 2By3 Sheet ;
1191:  !R[105]=AR[1]=200, 3By4 Sheet ;
1192:  !R[105]=AR[1]=410, 4By9 OFT ;
1193:  !R[105]=AR[1]=300, 5By7 Sheet ;
1194:  CALL JOB_VAR_SETUP(450) ;
1195:   ;
1196:  !--------------------------- ;
1197:  !Define Parameters for Job ;
1198:  !R[85] "INF_JAW_OFFSET"(Hgt) ;
1199:  R[85]=20    ;
1200:  !R[86] "INF_PICK_OFFSET" 50mm/sec ;
1201:  R[86]=0    ;
1202:  !R[87] "MAIN_LOAD_OFFSET" (PRELOA ;
1203:  R[87]=100    ;
1204:  !R[100] "GRIPPER_ID" 3 values ;
1205:  !If =100, ID Grippers Installed ;
1206:  !If =200, OD Grippers Installed ;
1207:  !If =300, OD 45 Degree Grippers ;
1208:  R[100]=200    ;
1209:  !--------------------------- ;
1210:   ;
1211:  !If using previous setup data ;
1212:  IF (R[71]=5649) THEN ;
1213:   ;
1214:  !--------------------------- ;
1215:  !1st: Height of Raw piece ;
1216:  R[190]=13.716    ;
1217:  !2nd: Height of Finish piece ;
1218:  R[191]=13.716    ;
1219:  !3rd: Infeed Height Offset ;
1220:  R[192]=55    ;
1221:  !4th: Outfeed Height Offset ;
1222:  R[193]=0    ;
1223:  !--------------------------- ;
1224:   ;
1225:  CALL CREATE_REG(R[190],R[191],R[192],R[193]) ;
1226:   ;
1227:  ENDIF ;
1228:   ;
1229:  !If new loading or offloading pos ;
1230:  !SET R[104] "IMPORT_LOADPOS" ;
1231:  !SET R[104]=1000, Otherwise NO ;
1232:  R[104]=1000    ;
1233:  IF (R[104]=1000) THEN ;
1234:  !R[260]=43, Preload Pos1 ;
1235:  !R[270]=44, Preload PosFinal ;
1236:  !R[300]=53, Offload PosFinal ;
1237:  !PR[43] Pre-Loading Pos1 ;
1238:  CALL CREATE_PR(43,165.28,(-63.404),200.524,145.664,89.044,143.591) ;
1239:  !PR[44] Final Loading Position ;
1240:  CALL CREATE_PR(44,165.457,(-63.614),212.699,145.745,89.043,143.668) ;
1241:  !PR[53] Pre Unloading Position ;
1242:  CALL CREATE_PR(53,(-127.177),96.912,209.866,(-109.535),(-89.592),111.616) ;
1243:  !PR[54] Final Unloading Position ;
1244:  CALL CREATE_PR(54,(-127.1),96.589,182.644,(-109.417),(-89.589),111.502) ;
1245:  !PR[56] assitant Unloading preses ;
1246:  CALL CREATE_PR(56,(-135.297),92.538,351.803,(-156.279),(-87.981),158.047) ;
1247:  !PR[57] assitant Unloading preses ;
1248:  CALL CREATE_PR(57,(-136.348),92.89,384.48,(-156.272),(-87.98),158.048) ;
1249:  !PR[58] assitant Unloading preses ;
1250:  CALL CREATE_PR(58,(-136.985),93.066,404.648,(-156.269),(-87.977),158.046) ;
1251:  ENDIF ;
1252:   ;
1253:  !---------------------------- ;
1254:  !SR[2] = "JOB_VAR_OD_GRIP" ;
1255:  !JOB_VAR_COMMON(R[103])'s value ;
1256:  !---------------------------- ;
1257:  !2By3 SR[2] INF, Max 18(Straight) ;
1258:  !R[103]=200 ;
1259:  !2By3 INF 45 Degree Diagonal Shif ;
1260:  !R[103]=210 ;
1261:  !---------------------------- ;
1262:  !3By4 SR[2] INF, Max 36(Straight) ;
1263:  !R[103]=250 ;
1264:  !3By4 INF 45 Degree Diagonal Shif ;
1265:  !R[103]=260 ;
1266:  !---------------------------- ;
1267:  !R[103] "JOB_PROFILE" Selection ;
1268:  R[103]=300    ;
1269:  CALL JOB_VAR_COMMON(R[103]) ;
1270:   ;
1271:  ENDIF ;
1272:   ;
1273:  JMP LBL[9999] ;
1274:   ;
1275:  !Job 1025649 Logic Ends ;
1276:  !--------------------------- ;
1277:   ;
1278:  LBL[5943] ;
1279:  !--------------------------- ;
1280:  !ADPTR ;
1281:  !Item 103365943, Rev A ;
1282:  !Last Modified: 2026-05-06 ;
1283:  !Modified by: Aaron ;
1284:  !8.3 IN Height ;
1285:  !3.15 IN ID, 4.38 IN OD 37.0 Lbs ;
1286:  !OD Jaw #2004 ;
1287:  !------------------------- ;
1288:  IF (R[70]=5943) THEN ;
1289:   ;
1290:  !Define Parameters for INF/OTF ;
1291:  !R[105]=AR[1]=100, 2By3 Sheet ;
1292:  !R[105]=AR[1]=200, 3By4 Sheet ;
1293:  !R[105]=AR[1]=300, 5By7 Sheet ;
1294:  CALL JOB_VAR_SETUP(100) ;
1295:   ;
1296:  !------------------------- ;
1297:  !Define Parameters for Job ;
1298:  R[1]=1    ;
1299:  R[67]=50    ;
1300:  R[2]=1    ;
1301:  R[139]=12    ;
1302:  R[3]=0    ;
1303:  R[4]=1    ;
1304:  R[85]=116.22    ;
1305:  R[86]=5    ;
1306:  R[87]=150    ;
1307:  R[95]=100    ;
1308:  R[110]=2004    ;
1309:  !CNC W-AXIS OFFSET ;
1310:  R[111]=((-16.06)) ;
1311:  !X-Compliance Push Bypass ;
1312:  F[6:OFF]=(OFF) ;
1313:  !--------------------------- ;
1314:  !R[100] "GRIPPER_ID" 3 values ;
1315:  !If =100, ID Grippers Installed ;
1316:  !If =200, OD Grippers Installed ;
1317:  !If =300, OD 45 Degree Grippers ;
1318:  R[100]=200    ;
1319:  !--------------------------- ;
1320:   ;
1321:  !If using previous setup data ;
1322:  IF (R[71]=5943) THEN ;
1323:   ;
1324:  !--------------------------- ;
1325:  R[190]=217.5    ;
1326:  R[191]=210.82    ;
1327:  R[192]=(-305)    ;
1328:  R[193]=(-170)    ;
1329:  !--------------------------- ;
1330:   ;
1331:   ;
1332:  CALL CREATE_REG(R[190],R[191],R[192],R[193]) ;
1333:   ;
1334:  ENDIF ;
1335:   ;
1336:  !If new loading or offloading pos ;
1337:  !SET R[104] "IMPORT_LOADPOS" ;
1338:  !SET R[104]=1000, Otherwise NO ;
1339:  R[104]=1000    ;
1340:  IF (R[104]=1000) THEN ;
1341:  !R[260]=43, Preload Pos1 ;
1342:  !R[270]=44, Preload PosFinal ;
1343:  !R[300]=53, Offload PosFinal ;
1344:  !PR[43] Pre-Loading Pos1 ;
1345:  CALL CREATE_PR(43,168.429,(-63.297),182.373,91.212,89.177,89.367) ;
1346:  !PR[44] Final Loading Position ;
1347:  CALL CREATE_PR(44,168.457,(-64.583),253.217,91.816,89.163,89.957) ;
1348:  !PR[53] Pre Unloading Position ;
1349:  CALL CREATE_PR(53,(-123.542),93.361,259.571,13.31,(-89.092),(-16.834)) ;
1350:  !PR[54] Final Unloading Position ;
1351:  CALL CREATE_PR(54,(-125.695),94.128,119.511,13.287,(-89.09),(-16.818)) ;
1352:  ENDIF ;
1353:   ;
1354:  !---------------------------- ;
1355:  !SR[2] = "JOB_VAR_OD_GRIP" ;
1356:  !JOB_VAR_COMMON(R[103])'s value ;
1357:  !---------------------------- ;
1358:  !2By3 SR[2] INF, Max 18(Straight) ;
1359:  !R[103]=200 ;
1360:  !2By3 INF 45 Degree Diagonal Shif ;
1361:  !R[103]=210 ;
1362:  !---------------------------- ;
1363:  !3By4 SR[2] INF, Max 36(Straight) ;
1364:  !R[103]=250 ;
1365:  !3By4 INF 45 Degree Diagonal Shif ;
1366:  !R[103]=260 ;
1367:  !---------------------------- ;
1368:  !R[103] "JOB_PROFILE" Selection ;
1369:  R[103]=200    ;
1370:  CALL JOB_VAR_COMMON(R[103]) ;
1371:   ;
1372:  ENDIF ;
1373:   ;
1374:  JMP LBL[9999] ;
1375:   ;
1376:  !Job 103365943 Logic Ends ;
1377:  !--------------------------- ;
1378:   ;
1379:  LBL[6372] ;
1380:  !--------------------------- ;
1381:  !Wedge ;
1382:  !Item 102906372 , Rev A ;
1383:  !Last Modified: 2022-12-13 ;
1384:  !Modified by: Tsuu ;
1385:  !1.89 IN Height ;
1386:  !1.61 IN ID, 3.15 IN OD ;
1387:  !OD Jaw # 2010 ;
1388:  !--------------------------- ;
1389:  IF (R[70]=6372) THEN ;
1390:  !Define Parameters for INF/OTF ;
1391:  !R[105]=AR[1]=100, 2By3 Sheet ;
1392:  !R[105]=AR[1]=200, 3By4 Sheet ;
1393:  !R[105]=AR[1]=300, 5By7 Sheet ;
1394:  CALL JOB_VAR_SETUP(200) ;
1395:   ;
1396:  !--------------------------- ;
1397:  !Define Parameters for Job ;
1398:  !R[85] "INF_JAW_OFFSET"(Hgt) ;
1399:  R[85]=42.75    ;
1400:  !R[86] "INF_PICK_OFFSET" 50mm/sec ;
1401:  R[86]=15    ;
1402:  !R[87] "MAIN_LOAD_OFFSET" (PRELOA ;
1403:  R[87]=100    ;
1404:  !R[100] "GRIPPER_ID" 3 values ;
1405:  !If =100, ID Grippers Installed ;
1406:  !If =200, OD Grippers Installed ;
1407:  !If =300, OD 45 Degree Grippers ;
1408:  R[100]=200    ;
1409:  !--------------------------- ;
1410:   ;
1411:  !If using previous setup data ;
1412:  IF (R[71]=6372) THEN ;
1413:   ;
1414:  !--------------------------- ;
1415:  !1st: Height of Raw piece ;
1416:  R[190]=51    ;
1417:  !2nd: Height of Finish piece ;
1418:  R[191]=48.006    ;
1419:  !3rd: Infeed Height Offset ;
1420:  R[192]=(-60)    ;
1421:  !4th: Outfeed Height Offset ;
1422:  R[193]=(-497)    ;
1423:  !--------------------------- ;
1424:   ;
1425:  CALL CREATE_REG(R[190],R[191],R[192],R[193]) ;
1426:   ;
1427:  ENDIF ;
1428:   ;
1429:  !If new loading or offloading pos ;
1430:  !SET R[104] "IMPORT_LOADPOS" ;
1431:  !SET R[104]=1000, Otherwise NO ;
1432:  R[104]=1000    ;
1433:  IF (R[104]=1000) THEN ;
1434:  !R[260]=43, Preload Pos1 ;
1435:  !R[270]=44, Preload PosFinal ;
1436:  !R[300]=53, Offload PosFinal ;
1437:  !PR[43] Pre-Loading Pos1 ;
1438:  CALL CREATE_PR(43,167.407,(-61.235),358.579,146.046,89.112,144.041) ;
1439:  !PR[44] Final Loading Position ;
1440:  CALL CREATE_PR(44,167.615,(-61.467),374.198,146.08,89.112,144.08) ;
1441:  !PR[53] Pre Unloading Position ;
1442:  CALL CREATE_PR(53,(-124.665),95.126,41.597,167.981,(-88.382),(-166.929)) ;
1443:  !PR[54] Final Unloading Position ;
1444:  CALL CREATE_PR(54,(-123.473),95.51,(-2.853),167.95,(-88.384),(-166.903)) ;
1445:  !PR[56] assitant Unloading preses ;
1446:  CALL CREATE_PR(56,(-131.536),105.713,233.177,173.746,(-88.233),(-175.647)) ;
1447:  !PR[57] assitant Unloading preses ;
1448:  CALL CREATE_PR(57,(-133.703),92.431,364.782,167.802,(-88.383),(-166.755)) ;
1449:  !PR[58] assitant Unloading preses ;
1450:  CALL CREATE_PR(58,(-133.703),92.431,364.782,167.804,(-88.383),(-166.755)) ;
1451:  ENDIF ;
1452:   ;
1453:  !---------------------------- ;
1454:  !SR[2] = "JOB_VAR_OD_GRIP" ;
1455:  !JOB_VAR_COMMON(R[103])'s value ;
1456:  !---------------------------- ;
1457:  !2By3 SR[2] INF, Max 18(Straight) ;
1458:  !R[103]=200 ;
1459:  !2By3 INF 45 Degree Diagonal Shif ;
1460:  !R[103]=210 ;
1461:  !---------------------------- ;
1462:  !3By4 SR[2] INF, Max 36(Straight) ;
1463:  !R[103]=250 ;
1464:  !3By4 INF 45 Degree Diagonal Shif ;
1465:  !R[103]=260 ;
1466:  !---------------------------- ;
1467:  !R[103] "JOB_PROFILE" Selection ;
1468:  R[103]=250    ;
1469:  CALL JOB_VAR_COMMON(R[103]) ;
1470:   ;
1471:  ENDIF ;
1472:   ;
1473:  JMP LBL[9999] ;
1474:   ;
1475:  !Job 102906372 Logic Ends ;
1476:  !--------------------------- ;
1477:   ;
1478:  LBL[6549] ;
1479:  !--------------------------- ;
1480:  !Mandrel ;
1481:  !Item 102666549 , Rev D ;
1482:  !Last Modified: 2022-04-29 ;
1483:  !Modified by: Tsuu ;
1484:  !11.79 IN Height ;
1485:  !1.0 IN ID, 1.94 IN OD ;
1486:  !ID Jaw # 2014 ;
1487:  !--------------------------- ;
1488:  IF (R[70]=6549) THEN ;
1489:  !Define Parameters for INF/OTF ;
1490:  !R[105]=AR[1]=100, 2By3 Sheet ;
1491:  !R[105]=AR[1]=200, 3By4 Sheet ;
1492:  !R[105]=AR[1]=210, 3By4 Sheet Man ;
1493:  !R[105]=AR[1]=300, 5By7 Sheet ;
1494:  CALL JOB_VAR_SETUP(210) ;
1495:   ;
1496:  !--------------------------- ;
1497:  !Define Parameters for Job ;
1498:  !R[85] "INF_JAW_OFFSET"(Hgt) ;
1499:  R[85]=30    ;
1500:  !R[86] "INF_PICK_OFFSET" 50mm/sec ;
1501:  R[86]=10    ;
1502:  !R[87] "MAIN_LOAD_OFFSET" (PRELOA ;
1503:  R[87]=0    ;
1504:  !R[100] "GRIPPER_ID" 3 values ;
1505:  !If =100, ID Grippers Installed ;
1506:  !If =200, OD Grippers Installed ;
1507:  !If =300, OD 45 Degree Grippers ;
1508:  R[100]=200    ;
1509:  !--------------------------- ;
1510:   ;
1511:  !If using previous setup data ;
1512:  IF (R[71]=6549) THEN ;
1513:   ;
1514:  !--------------------------- ;
1515:  !1st: Height of Raw piece ;
1516:  R[190]=303.5    ;
1517:  !2nd: Height of Finish piece ;
1518:  R[191]=299.459    ;
1519:  !3rd: Infeed Height Offset ;
1520:  R[192]=(-485)    ;
1521:  !4th: Outfeed Height Offset ;
1522:  R[193]=(-346)    ;
1523:  !--------------------------- ;
1524:   ;
1525:  CALL CREATE_REG(R[190],R[191],R[192],R[193]) ;
1526:   ;
1527:  ENDIF ;
1528:   ;
1529:  !If new loading or offloading pos ;
1530:  !SET R[104] "IMPORT_LOADPOS" ;
1531:  !SET R[104]=1000, Otherwise NO ;
1532:  R[104]=1000    ;
1533:  IF (R[104]=1000) THEN ;
1534:  !R[260]=43, Preload Pos1 ;
1535:  !R[270]=44, Preload PosFinal ;
1536:  !R[300]=53, Offload PosFinal ;
1537:  !PR[43] Pre-Loading Pos1 ;
1538:  CALL CREATE_PR(43,163.336,(-59.078),66.326,122.498,89.025,120.434) ;
1539:  !PR[44] Final Loading Position ;
1540:  CALL CREATE_PR(44,165.548,(-60.288),161.604,138.028,88.79,135.951) ;
1541:  !PR[53] Pre Unloading Position ;
1542:  CALL CREATE_PR(53,(-126.684),95.87,26.133,170.552,(-88.453),(-172.384)) ;
1543:  !PR[54] Final Unloading Position ;
1544:  CALL CREATE_PR(54,(-125.869),95.755,(-4.385),170.71,(-88.454),(-172.531)) ;
1545:  !PR[56] assitant Unloading preses ;
1546:  CALL CREATE_PR(56,(-127.606),95.642,60.969,170.577,(-88.453),(-172.403)) ;
1547:  !PR[57] assitant Unloading preses ;
1548:  CALL CREATE_PR(57,(-129.985),95.23,150.815,170.613,(-88.45),(-172.434)) ;
1549:  !PR[58] assitant Unloading preses ;
1550:  CALL CREATE_PR(58,(-132.052),94.793,229.549,170.647,(-88.449),(-172.464)) ;
1551:  !PR[59] assitant Unloading preses ;
1552:  CALL CREATE_PR(59,82.373,234.687,398.527,(-91.753),0,88.068) ;
1553:  ENDIF ;
1554:   ;
1555:  !---------------------------- ;
1556:  !SR[2] = "JOB_VAR_OD_GRIP" ;
1557:  !JOB_VAR_COMMON(R[103])'s value ;
1558:  !---------------------------- ;
1559:  !2By3 SR[2] INF, Max 18(Straight) ;
1560:  !R[103]=200 ;
1561:  !2By3 INF 45 Degree Diagonal Shif ;
1562:  !R[103]=210 ;
1563:  !---------------------------- ;
1564:  !3By4 SR[2] INF, Max 36(Straight) ;
1565:  !R[103]=250 ;
1566:  !3By4 INF Mandrel, 2 Trays ;
1567:  !R[103]=260 ;
1568:  !---------------------------- ;
1569:  !R[103] "JOB_PROFILE" Selection ;
1570:  R[103]=260    ;
1571:  CALL JOB_VAR_COMMON(R[103]) ;
1572:   ;
1573:  ENDIF ;
1574:   ;
1575:  JMP LBL[9999] ;
1576:   ;
1577:  !Job 102666549 Logic Ends ;
1578:  !--------------------------- ;
1579:   ;
1580:  LBL[6588] ;
1581:  !------------------------- ;
1582:  !Cup-Spring, NFI ;
1583:  !Item 1026588 ,Rev A ;
1584:  !Last Modified: 2024-09-24 ;
1585:  !Modified by: Tsuu ;
1586:  !0.272 IN Hgt ;
1587:  !0.220 IN ID, 0.884 IN OD ;
1588:  !OD Jaw #1036 ;
1589:  !--------------------------- ;
1590:  IF (R[70]=6588) THEN ;
1591:  !Define Parameters for INF/OTF ;
1592:  !R[105]=AR[1]=100, 2By3 Sheet ;
1593:  !R[105]=AR[1]=200, 3By4 Sheet ;
1594:  !R[105]=AR[1]=410, 4By9 OFT ;
1595:  !R[105]=AR[1]=300, 5By7 Sheet ;
1596:  !R[105]=AR[1]=470, 6By8 OFT ;
1597:  !R[105]=AR[1]=450, 8By6 OFT ;
1598:  CALL JOB_VAR_SETUP(470) ;
1599:   ;
1600:  !--------------------------- ;
1601:  !Define Parameters for Job ;
1602:  !R[1] JAW PUSH ;
1603:  R[1]=0    ;
1604:  !R[2] NEVER DROP ;
1605:  R[2]=0    ;
1606:  !R[3] BAR FEED ;
1607:  R[3]=1    ;
1608:  !R[4] HEAVY PART ;
1609:  R[4]=0    ;
1610:  !R[85] "INF_JAW_OFFSET"(Hgt) ;
1611:  R[85]=20    ;
1612:  !R[86] "INF_PICK_OFFSET" 50mm/sec ;
1613:  R[86]=0    ;
1614:  !R[87] "MAIN_LOAD_OFFSET" (PRELOA ;
1615:  R[87]=100    ;
1616:  !R[100] "GRIPPER_ID" 3 values ;
1617:  !If =100, ID Grippers Installed ;
1618:  !If =200, OD Grippers Installed ;
1619:  !If =300, OD 45 Degree Grippers ;
1620:  R[100]=200    ;
1621:  !--------------------------- ;
1622:   ;
1623:  !If using previous setup data ;
1624:  IF (R[71]=6588) THEN ;
1625:   ;
1626:  !--------------------------- ;
1627:  !1st: Height of Raw piece ;
1628:  R[190]=7.45    ;
1629:  !2nd: Height of Finish piece ;
1630:  R[191]=7.45    ;
1631:  !3rd: Infeed Height Offset ;
1632:  R[192]=55    ;
1633:  !4th: Outfeed Height Offset ;
1634:  R[193]=(-50)    ;
1635:  !--------------------------- ;
1636:   ;
1637:  CALL CREATE_REG(R[190],R[191],R[192],R[193]) ;
1638:   ;
1639:  ENDIF ;
1640:   ;
1641:  !If new loading or offloading pos ;
1642:  !SET R[104] "IMPORT_LOADPOS" ;
1643:  !SET R[104]=1000, Otherwise NO ;
1644:  R[104]=1000    ;
1645:  IF (R[104]=1000) THEN ;
1646:  !R[260]=43, Preload Pos1 ;
1647:  !R[270]=44, Preload PosFinal ;
1648:  !R[300]=53, Offload PosFinal ;
1649:  !PR[43] Pre-Loading Pos1 ;
1650:  CALL CREATE_PR(43,165.28,(-63.404),200.524,145.664,89.044,143.591) ;
1651:  !PR[44] Final Loading Position ;
1652:  CALL CREATE_PR(44,165.457,(-63.614),212.699,145.745,89.043,143.668) ;
1653:  !PR[53] Pre Unloading Position ;
1654:  CALL CREATE_PR(53,(-126.139),96.136,126.303,(-97.393),(-89.556),99.662) ;
1655:  !PR[54] Final Unloading Position ;
1656:  CALL CREATE_PR(54,(-126.161),96.188,117.696,(-97.131),(-89.557),99.392) ;
1657:  ENDIF ;
1658:   ;
1659:  !---------------------------- ;
1660:  !SR[2] = "JOB_VAR_OD_GRIP" ;
1661:  !JOB_VAR_COMMON(R[103])'s value ;
1662:  !---------------------------- ;
1663:  !2By3 SR[2] INF, Max 18(Straight) ;
1664:  !R[103]=200 ;
1665:  !2By3 INF 45 Degree Diagonal Shif ;
1666:  !R[103]=210 ;
1667:  !---------------------------- ;
1668:  !3By4 SR[2] INF, Max 36(Straight) ;
1669:  !R[103]=250 ;
1670:  !3By4 INF 45 Degree Diagonal Shif ;
1671:  !R[103]=260 ;
1672:  !---------------------------- ;
1673:  !R[103] "JOB_PROFILE" Selection ;
1674:  R[103]=320    ;
1675:  CALL JOB_VAR_COMMON(R[103]) ;
1676:   ;
1677:  ENDIF ;
1678:   ;
1679:  JMP LBL[9999] ;
1680:   ;
1681:  !Job 1026588 Logic Ends ;
1682:  !--------------------------- ;
1683:   ;
1684:  LBL[6617] ;
1685:  !------------------------- ;
1686:  !CARTRIDGE NFI AL ;
1687:  !Item 1026617 ,Rev A ;
1688:  !Last Modified: 2024-11-19 ;
1689:  !Modified by: Tsuu ;
1690:  !0.625 IN Hgt ;
1691:  !1.0 IN ID, 2.250 IN OD ;
1692:  !OD Jaw #2012 ;
1693:  !--------------------------- ;
1694:  IF (R[70]=6617) THEN ;
1695:  !Define Parameters for INF/OTF ;
1696:  !R[105]=AR[1]=100, 2By3 Sheet ;
1697:  !R[105]=AR[1]=200, 3By4 Sheet ;
1698:  !R[105]=AR[1]=410, 4By9 OFT ;
1699:  !R[105]=AR[1]=300, 5By7 Sheet ;
1700:  CALL JOB_VAR_SETUP(470) ;
1701:   ;
1702:  !--------------------------- ;
1703:  !Define Parameters for Job ;
1704:  R[1]=0    ;
1705:  R[67]=20    ;
1706:  R[2]=0    ;
1707:  R[139]=20    ;
1708:  R[3]=1    ;
1709:  R[4]=0    ;
1710:  !R[85] "INF_JAW_OFFSET"(Hgt) ;
1711:  R[85]=20    ;
1712:  !R[86] "INF_PICK_OFFSET" 50mm/sec ;
1713:  R[86]=0    ;
1714:  !R[87] "MAIN_LOAD_OFFSET" (PRELOA ;
1715:  R[87]=100    ;
1716:  !R[100] "GRIPPER_ID" 3 values ;
1717:  !If =100, ID Grippers Installed ;
1718:  !If =200, OD Grippers Installed ;
1719:  !If =300, OD 45 Degree Grippers ;
1720:  R[100]=200    ;
1721:  !--------------------------- ;
1722:   ;
1723:  !If using previous setup data ;
1724:  IF (R[71]=6617) THEN ;
1725:   ;
1726:  !--------------------------- ;
1727:  !1st: Height of Raw piece ;
1728:  R[190]=45.72    ;
1729:  !2nd: Height of Finish piece ;
1730:  R[191]=40.64    ;
1731:  !3rd: Infeed Height Offset ;
1732:  R[192]=55    ;
1733:  !4th: Outfeed Height Offset ;
1734:  R[193]=(-110)    ;
1735:  !--------------------------- ;
1736:   ;
1737:  CALL CREATE_REG(R[190],R[191],R[192],R[193]) ;
1738:   ;
1739:  ENDIF ;
1740:   ;
1741:  !If new loading or offloading pos ;
1742:  !SET R[104] "IMPORT_LOADPOS" ;
1743:  !SET R[104]=1000, Otherwise NO ;
1744:  R[104]=1000    ;
1745:  IF (R[104]=1000) THEN ;
1746:  !R[260]=43, Preload Pos1 ;
1747:  !R[270]=44, Preload PosFinal ;
1748:  !R[300]=53, Offload PosFinal ;
1749:  !PR[43] Pre-Loading Pos1 ;
1750:  CALL CREATE_PR(43,165.28,(-63.404),200.524,145.664,89.044,143.591) ;
1751:  !PR[44] Final Loading Position ;
1752:  CALL CREATE_PR(44,165.457,(-63.614),212.699,145.745,89.043,143.668) ;
1753:  !PR[53] Pre Unloading Position ;
1754:  CALL CREATE_PR(53,(-123.662),96.487,41.452,(-24.867),(-89.839),27.065) ;
1755:  !PR[54] Final Unloading Position ;
1756:  CALL CREATE_PR(54,(-123.757),96.523,16.909,(-25.018),(-89.837),27.212) ;
1757:  !PR[56] assitant Unloading preses ;
1758:  CALL CREATE_PR(56,(-135.297),92.538,351.803,(-156.279),(-87.981),158.047) ;
1759:  !PR[57] assitant Unloading preses ;
1760:  CALL CREATE_PR(57,(-136.348),92.89,384.48,(-156.272),(-87.98),158.048) ;
1761:  !PR[58] assitant Unloading preses ;
1762:  CALL CREATE_PR(58,(-136.985),93.066,404.648,(-156.269),(-87.977),158.046) ;
1763:  ENDIF ;
1764:   ;
1765:  !---------------------------- ;
1766:  !SR[2] = "JOB_VAR_OD_GRIP" ;
1767:  !JOB_VAR_COMMON(R[103])'s value ;
1768:  !---------------------------- ;
1769:  !2By3 SR[2] INF, Max 18(Straight) ;
1770:  !R[103]=200 ;
1771:  !2By3 INF 45 Degree Diagonal Shif ;
1772:  !R[103]=210 ;
1773:  !---------------------------- ;
1774:  !3By4 SR[2] INF, Max 36(Straight) ;
1775:  !R[103]=250 ;
1776:  !3By4 INF 45 Degree Diagonal Shif ;
1777:  !R[103]=260 ;
1778:  !---------------------------- ;
1779:  !R[103] "JOB_PROFILE" Selection ;
1780:  R[103]=280    ;
1781:  CALL JOB_VAR_COMMON(R[103]) ;
1782:   ;
1783:  ENDIF ;
1784:   ;
1785:  JMP LBL[9999] ;
1786:   ;
1787:  !Job 1026617 Logic Ends ;
1788:  !--------------------------- ;
1789:   ;
1790:  LBL[6754] ;
1791:  !------------------------- ;
1792:  !Rapid Ball ;
1793:  !Item 102606754 , Rev xxx ;
1794:  !Last Modified: 2021-06-15 ;
1795:  !Modified by: Tsuu ;
1796:  !1.6 IN Height ;
1797:  !0 ID, 1.6 OD ;
1798:  !OD Jaw #3003 ;
1799:  !--------------------------- ;
1800:  IF (R[70]=6754) THEN ;
1801:  !Define Parameters for INF/OTF ;
1802:  !R[105]=AR[1]=100, 2By3 Sheet ;
1803:  !R[105]=AR[1]=200, 3By4 Sheet ;
1804:  !R[105]=AR[1]=300, 5By7 Sheet ;
1805:  CALL JOB_VAR_SETUP(400) ;
1806:   ;
1807:  !--------------------------- ;
1808:  !Define Parameters for Job ;
1809:  !R[85] "INF_JAW_OFFSET"(Hgt) ;
1810:  R[85]=97    ;
1811:  !R[86] "INF_PICK_OFFSET" 50mm/sec ;
1812:  R[86]=0    ;
1813:  !R[87] "MAIN_LOAD_OFFSET" (PRELOA ;
1814:  R[87]=100    ;
1815:  !R[100] "GRIPPER_ID" 3 values ;
1816:  !If =100, ID Grippers Installed ;
1817:  !If =200, OD Grippers Installed ;
1818:  !If =300, OD 45 Degree Grippers ;
1819:  R[100]=200    ;
1820:  !--------------------------- ;
1821:   ;
1822:  !If using previous setup data ;
1823:  IF (R[71]=6754) THEN ;
1824:   ;
1825:  !--------------------------- ;
1826:  !1st: Height of Raw piece ;
1827:  R[190]=45.72    ;
1828:  !2nd: Height of Finish piece ;
1829:  R[191]=40.64    ;
1830:  !3rd: Infeed Height Offset ;
1831:  R[192]=55    ;
1832:  !4th: Outfeed Height Offset ;
1833:  R[193]=90    ;
1834:  !--------------------------- ;
1835:   ;
1836:  CALL CREATE_REG(R[190],R[191],R[192],R[193]) ;
1837:   ;
1838:  ENDIF ;
1839:   ;
1840:  !If new loading or offloading pos ;
1841:  !SET R[104] "IMPORT_LOADPOS" ;
1842:  !SET R[104]=1000, Otherwise NO ;
1843:  R[104]=1000    ;
1844:  IF (R[104]=1000) THEN ;
1845:  !R[260]=43, Preload Pos1 ;
1846:  !R[270]=44, Preload PosFinal ;
1847:  !R[300]=53, Offload PosFinal ;
1848:  !PR[43] Pre-Loading Pos1 ;
1849:  CALL CREATE_PR(43,165.28,(-63.404),200.524,145.664,89.044,143.591) ;
1850:  !PR[44] Final Loading Position ;
1851:  CALL CREATE_PR(44,165.457,(-63.614),212.699,145.745,89.043,143.668) ;
1852:  !PR[53] Pre Unloading Position ;
1853:  CALL CREATE_PR(53,(-133.516),91.907,296.601,(-156.3),(-87.984),158.064) ;
1854:  !PR[54] Final Unloading Position ;
1855:  CALL CREATE_PR(54,(-132.217),91.476,256.294,(-156.321),(-87.987),158.078) ;
1856:  !PR[56] assitant Unloading preses ;
1857:  CALL CREATE_PR(56,(-135.297),92.538,351.803,(-156.279),(-87.981),158.047) ;
1858:  !PR[57] assitant Unloading preses ;
1859:  CALL CREATE_PR(57,(-136.348),92.89,384.48,(-156.272),(-87.98),158.048) ;
1860:  !PR[58] assitant Unloading preses ;
1861:  CALL CREATE_PR(58,(-136.985),93.066,404.648,(-156.269),(-87.977),158.046) ;
1862:  ENDIF ;
1863:   ;
1864:  !---------------------------- ;
1865:  !SR[2] = "JOB_VAR_OD_GRIP" ;
1866:  !JOB_VAR_COMMON(R[103])'s value ;
1867:  !---------------------------- ;
1868:  !2By3 SR[2] INF, Max 18(Straight) ;
1869:  !R[103]=200 ;
1870:  !2By3 INF 45 Degree Diagonal Shif ;
1871:  !R[103]=210 ;
1872:  !---------------------------- ;
1873:  !3By4 SR[2] INF, Max 36(Straight) ;
1874:  !R[103]=250 ;
1875:  !3By4 INF 45 Degree Diagonal Shif ;
1876:  !R[103]=260 ;
1877:  !---------------------------- ;
1878:  !R[103] "JOB_PROFILE" Selection ;
1879:  R[103]=270    ;
1880:  CALL JOB_VAR_COMMON(R[103]) ;
1881:   ;
1882:  ENDIF ;
1883:   ;
1884:  JMP LBL[9999] ;
1885:   ;
1886:  !Job 102606754 Logic Ends ;
1887:  !--------------------------- ;
1888:   ;
1889:  LBL[6755] ;
1890:  !--------------------------- ;
1891:  !Rapid Ball ;
1892:  !Item 102606755 , Rev xxx ;
1893:  !Last Modified: 2021-02-23 ;
1894:  !Modified by: Tsuu ;
1895:  !2.0 IN Height ;
1896:  !0 ID, 2.0 OD ;
1897:  !OD Jaw #3001 ;
1898:  !--------------------------- ;
1899:  IF (R[70]=6755) THEN ;
1900:  !Define Parameters for INF/OTF ;
1901:  !R[105]=AR[1]=100, 2By3 Sheet ;
1902:  !R[105]=AR[1]=200, 3By4 Sheet ;
1903:  !R[105]=AR[1]=300, 5By7 Sheet ;
1904:  CALL JOB_VAR_SETUP(400) ;
1905:   ;
1906:  !--------------------------- ;
1907:  !Define Parameters for Job ;
1908:  !R[85] "INF_JAW_OFFSET"(Hgt) ;
1909:  R[85]=97    ;
1910:  !R[86] "INF_PICK_OFFSET" 50mm/sec ;
1911:  R[86]=0    ;
1912:  !R[87] "MAIN_LOAD_OFFSET" (PRELOA ;
1913:  R[87]=100    ;
1914:  !R[100] "GRIPPER_ID" 3 values ;
1915:  !If =100, ID Grippers Installed ;
1916:  !If =200, OD Grippers Installed ;
1917:  !If =300, OD 45 Degree Grippers ;
1918:  R[100]=200    ;
1919:  !--------------------------- ;
1920:   ;
1921:  !If using previous setup data ;
1922:  IF (R[71]=6755) THEN ;
1923:   ;
1924:  !--------------------------- ;
1925:  !1st: Height of Raw piece ;
1926:  R[190]=56.15    ;
1927:  !2nd: Height of Finish piece ;
1928:  R[191]=50    ;
1929:  !3rd: Infeed Height Offset ;
1930:  R[192]=(-96)    ;
1931:  !4th: Outfeed Height Offset ;
1932:  R[193]=(-46.5)    ;
1933:  !--------------------------- ;
1934:   ;
1935:  CALL CREATE_REG(R[190],R[191],R[192],R[193]) ;
1936:   ;
1937:  ENDIF ;
1938:   ;
1939:  !If new loading or offloading pos ;
1940:  !SET R[104] "IMPORT_LOADPOS" ;
1941:  !SET R[104]=1000, Otherwise NO ;
1942:  R[104]=1000    ;
1943:  IF (R[104]=1000) THEN ;
1944:  !R[260]=43, Preload Pos1 ;
1945:  !R[270]=44, Preload PosFinal ;
1946:  !R[300]=53, Offload PosFinal ;
1947:  !PR[43] Pre-Loading Pos1 ;
1948:  CALL CREATE_PR(43,168.835,(-63.534),347.629,158.268,89.347,156.235) ;
1949:  !PR[44] Final Loading Position ;
1950:  CALL CREATE_PR(44,168.927,(-63.781),356.006,158.173,89.348,156.13) ;
1951:  !PR[53] Pre Unloading Position ;
1952:  CALL CREATE_PR(53,(-129.883),93.702,179.02,170.509,(-88.382),(-168.991)) ;
1953:  !PR[54] Final Unloading Position ;
1954:  CALL CREATE_PR(54,(-128.536),94.044,130.257,170.547,(-88.382),(-169.034)) ;
1955:  !PR[56] assitant Unloading preses ;
1956:  CALL CREATE_PR(56,(-131.536),105.713,233.177,173.746,(-88.233),(-175.647)) ;
1957:  !PR[57] assitant Unloading preses ;
1958:  CALL CREATE_PR(57,(-131.536),105.713,233.177,173.746,(-88.233),(-175.647)) ;
1959:  !PR[58] assitant Unloading preses ;
1960:  CALL CREATE_PR(58,(-131.536),105.713,233.177,173.746,(-88.233),(-175.647)) ;
1961:  ENDIF ;
1962:   ;
1963:  !---------------------------- ;
1964:  !SR[2] = "JOB_VAR_OD_GRIP" ;
1965:  !JOB_VAR_COMMON(R[103])'s value ;
1966:  !---------------------------- ;
1967:  !2By3 SR[2] INF, Max 18(Straight) ;
1968:  !R[103]=200 ;
1969:  !2By3 INF 45 Degree Diagonal Shif ;
1970:  !R[103]=210 ;
1971:  !---------------------------- ;
1972:  !3By4 SR[2] INF, Max 36(Straight) ;
1973:  !R[103]=250 ;
1974:  !3By4 INF 45 Degree Diagonal Shif ;
1975:  !R[103]=260 ;
1976:  !---------------------------- ;
1977:  !R[103] "JOB_PROFILE" Selection ;
1978:  R[103]=270    ;
1979:  CALL JOB_VAR_COMMON(R[103]) ;
1980:   ;
1981:  ENDIF ;
1982:   ;
1983:  JMP LBL[9999] ;
1984:   ;
1985:  !Job 102606755 Logic Ends ;
1986:  !--------------------------- ;
1987:   ;
1988:  LBL[6756] ;
1989:  !--------------------------- ;
1990:  !Rapid Ball ;
1991:  !Item 102606756 , Rev xxx ;
1992:  !Last Modified: 2021-02-23 ;
1993:  !Modified by: Tsuu ;
1994:  !2.0 IN Height ;
1995:  !0 ID, 2.0 OD ;
1996:  !OD Jaw #3001 ;
1997:  !--------------------------- ;
1998:  IF (R[70]=6756) THEN ;
1999:  !Define Parameters for INF/OTF ;
2000:  !R[105]=AR[1]=100, 2By3 Sheet ;
2001:  !R[105]=AR[1]=200, 3By4 Sheet ;
2002:  !R[105]=AR[1]=300, 5By7 Sheet ;
2003:  CALL JOB_VAR_SETUP(400) ;
2004:   ;
2005:  !--------------------------- ;
2006:  !Define Parameters for Job ;
2007:  !R[85] "INF_JAW_OFFSET"(Hgt) ;
2008:  R[85]=97    ;
2009:  !R[86] "INF_PICK_OFFSET" 50mm/sec ;
2010:  R[86]=0    ;
2011:  !R[87] "MAIN_LOAD_OFFSET" (PRELOA ;
2012:  R[87]=100    ;
2013:  !R[100] "GRIPPER_ID" 3 values ;
2014:  !If =100, ID Grippers Installed ;
2015:  !If =200, OD Grippers Installed ;
2016:  !If =300, OD 45 Degree Grippers ;
2017:  R[100]=200    ;
2018:  !--------------------------- ;
2019:   ;
2020:  !If using previous setup data ;
2021:  IF (R[71]=6756) THEN ;
2022:   ;
2023:  !--------------------------- ;
2024:  !1st: Height of Raw piece ;
2025:  R[190]=56.15    ;
2026:  !2nd: Height of Finish piece ;
2027:  R[191]=50    ;
2028:  !3rd: Infeed Height Offset ;
2029:  R[192]=30    ;
2030:  !4th: Outfeed Height Offset ;
2031:  R[193]=82    ;
2032:  !--------------------------- ;
2033:   ;
2034:  CALL CREATE_REG(R[190],R[191],R[192],R[193]) ;
2035:   ;
2036:  ENDIF ;
2037:   ;
2038:  !If new loading or offloading pos ;
2039:  !SET R[104] "IMPORT_LOADPOS" ;
2040:  !SET R[104]=1000, Otherwise NO ;
2041:  R[104]=1000    ;
2042:  IF (R[104]=1000) THEN ;
2043:  !R[260]=43, Preload Pos1 ;
2044:  !R[270]=44, Preload PosFinal ;
2045:  !R[300]=53, Offload PosFinal ;
2046:  !PR[43] Pre-Loading Pos1 ;
2047:  CALL CREATE_PR(43,165.039,(-63.364),217.768,147.644,89.12,145.562) ;
2048:  !PR[44] Final Loading Position ;
2049:  CALL CREATE_PR(44,165.541,(-63.639),227.037,147.595,89.12,145.505) ;
2050:  !PR[53] Pre Unloading Position ;
2051:  CALL CREATE_PR(53,(-133.272),96.039,284.872,(-155.571),(-87.952),157.289) ;
2052:  !PR[54] Final Unloading Position ;
2053:  CALL CREATE_PR(54,(-132.253),95.709,253.312,(-155.638),(-87.954),157.353) ;
2054:  !PR[56] assitant Unloading preses ;
2055:  CALL CREATE_PR(56,(-134.36),96.418,318.618,(-155.552),(-87.949),157.274) ;
2056:  !PR[57] assitant Unloading preses ;
2057:  CALL CREATE_PR(57,(-135.431),96.699,352.37,(-155.498),(-87.943),157.231) ;
2058:  !PR[58] assitant Unloading preses ;
2059:  CALL CREATE_PR(58,(-135.431),96.699,352.37,(-155.498),(-87.943),157.231) ;
2060:  ENDIF ;
2061:   ;
2062:  !---------------------------- ;
2063:  !SR[2] = "JOB_VAR_OD_GRIP" ;
2064:  !JOB_VAR_COMMON(R[103])'s value ;
2065:  !---------------------------- ;
2066:  !2By3 SR[2] INF, Max 18(Straight) ;
2067:  !R[103]=200 ;
2068:  !2By3 INF 45 Degree Diagonal Shif ;
2069:  !R[103]=210 ;
2070:  !---------------------------- ;
2071:  !3By4 SR[2] INF, Max 36(Straight) ;
2072:  !R[103]=250 ;
2073:  !3By4 INF 45 Degree Diagonal Shif ;
2074:  !R[103]=260 ;
2075:  !---------------------------- ;
2076:  !R[103] "JOB_PROFILE" Selection ;
2077:  R[103]=270    ;
2078:  CALL JOB_VAR_COMMON(R[103]) ;
2079:   ;
2080:  ENDIF ;
2081:   ;
2082:  JMP LBL[9999] ;
2083:   ;
2084:  !Job 102606756 Logic Ends ;
2085:  !--------------------------- ;
2086:   ;
2087:  LBL[7062] ;
2088:  !--------------------------- ;
2089:  !Rapid Ball ;
2090:  !Item 102757062 , Rev D ;
2091:  !Last Modified: 2022-09-13 ;
2092:  !Modified by: Tsuu ;
2093:  !2.45 IN Height ;
2094:  !0 ID, 2.45 IN OD ;
2095:  !OD Jaw #3001 ;
2096:  !--------------------------- ;
2097:  IF (R[70]=7062) THEN ;
2098:  !Define Parameters for INF/OTF ;
2099:  !R[105]=AR[1]=100, 2By3 Sheet ;
2100:  !R[105]=AR[1]=200, 3By4 Sheet ;
2101:  !R[105]=AR[1]=300, 5By7 Sheet ;
2102:  !R[105]=AR[1]=400, 4By6 Sheet ;
2103:  CALL JOB_VAR_SETUP(450) ;
2104:   ;
2105:  !--------------------------- ;
2106:  !Define Parameters for Job ;
2107:  !R[85] "INF_JAW_OFFSET"(Hgt) ;
2108:  R[85]=97    ;
2109:  !R[86] "INF_PICK_OFFSET" 50mm/sec ;
2110:  R[86]=0    ;
2111:  !R[87] "MAIN_LOAD_OFFSET" (PRELOA ;
2112:  R[87]=0    ;
2113:  !R[100] "GRIPPER_ID" 3 values ;
2114:  !If =100, ID Grippers Installed ;
2115:  !If =200, OD Grippers Installed ;
2116:  !If =300, OD 45 Degree Grippers ;
2117:  R[100]=200    ;
2118:  !--------------------------- ;
2119:   ;
2120:  !If using previous setup data ;
2121:  IF (R[71]=7062) THEN ;
2122:   ;
2123:  !--------------------------- ;
2124:  !1st: Height of Raw piece ;
2125:  R[190]=68.55    ;
2126:  !2nd: Height of Finish piece ;
2127:  R[191]=62.15    ;
2128:  !3rd: Infeed Height Offset ;
2129:  R[192]=(-85)    ;
2130:  !4th: Outfeed Height Offset ;
2131:  R[193]=(-30)    ;
2132:  !--------------------------- ;
2133:   ;
2134:  CALL CREATE_REG(R[190],R[191],R[192],R[193]) ;
2135:   ;
2136:  ENDIF ;
2137:   ;
2138:  !If new loading or offloading pos ;
2139:  !SET R[104] "IMPORT_LOADPOS" ;
2140:  !SET R[104]=1000, Otherwise NO ;
2141:  R[104]=1000    ;
2142:  IF (R[104]=1000) THEN ;
2143:  !R[260]=43, Preload Pos1 ;
2144:  !R[270]=44, Preload PosFinal ;
2145:  !R[300]=53, Offload PosFinal ;
2146:  !PR[43] Pre-Loading Pos1 ;
2147:  CALL CREATE_PR(43,168.763,(-63.729),319.101,149.882,89.211,147.864) ;
2148:  !PR[44] Final Loading Position ;
2149:  CALL CREATE_PR(44,168.912,(-63.908),331.315,149.906,89.21,147.882) ;
2150:  !PR[53] Pre Unloading Position ;
2151:  CALL CREATE_PR(53,(-130.417),91.762,201.726,170.612,(-88.383),(-169.064)) ;
2152:  !PR[54] Final Unloading Position ;
2153:  CALL CREATE_PR(54,(-129.142),92.087,155.419,170.61,(-88.383),(-169.064)) ;
2154:  !PR[56] assitant Unloading preses ;
2155:  CALL CREATE_PR(56,(-131.536),105.713,233.177,173.746,(-88.233),(-175.647)) ;
2156:  !PR[57] assitant Unloading preses ;
2157:  CALL CREATE_PR(57,(-131.536),105.713,233.177,173.746,(-88.233),(-175.647)) ;
2158:  !PR[58] assitant Unloading preses ;
2159:  CALL CREATE_PR(58,(-131.536),105.713,233.177,173.746,(-88.233),(-175.647)) ;
2160:  ENDIF ;
2161:   ;
2162:  !---------------------------- ;
2163:  !SR[2] = "JOB_VAR_OD_GRIP" ;
2164:  !JOB_VAR_COMMON(R[103])'s value ;
2165:  !---------------------------- ;
2166:  !2By3 SR[2] INF, Max 18(Straight) ;
2167:  !R[103]=200 ;
2168:  !2By3 INF 45 Degree Diagonal Shif ;
2169:  !R[103]=210 ;
2170:  !---------------------------- ;
2171:  !3By4 SR[2] INF, Max 36(Straight) ;
2172:  !R[103]=250 ;
2173:  !3By4 INF 45 Degree Diagonal Shif ;
2174:  !R[103]=260 ;
2175:  !4By6 INF OD-GRIP, Max 144 piece ;
2176:  !R[103]=270 ;
2177:  !4By6 INF OD-GRIP, Max 144 piece ;
2178:  !R[103]=280 ;
2179:  !---------------------------- ;
2180:  !R[103] "JOB_PROFILE" Selection ;
2181:  R[103]=280    ;
2182:  CALL JOB_VAR_COMMON(R[103]) ;
2183:   ;
2184:  ENDIF ;
2185:   ;
2186:  JMP LBL[9999] ;
2187:   ;
2188:  !Job 102757062 Logic Ends ;
2189:  !--------------------------- ;
2190:   ;
2191:  LBL[7436] ;
2192:  !------------------------- ;
2193:  !Rapid Ball ;
2194:  !Item 102577436 , Rev B ;
2195:  !Last Modified: 2023-01-03 ;
2196:  !Modified by: Tsuu ;
2197:  !1.36 IN Height ;
2198:  !0 ID, 1.360 OD ;
2199:  !OD Jaw #3003 ;
2200:  !--------------------------- ;
2201:  IF (R[70]=7436) THEN ;
2202:  !Define Parameters for INF/OTF ;
2203:  !R[105]=AR[1]=100, 2By3 Sheet ;
2204:  !R[105]=AR[1]=200, 3By4 Sheet ;
2205:  !R[105]=AR[1]=300, 5By7 Sheet ;
2206:  CALL JOB_VAR_SETUP(400) ;
2207:   ;
2208:  !--------------------------- ;
2209:  !Define Parameters for Job ;
2210:  !R[85] "INF_JAW_OFFSET"(Hgt) ;
2211:  R[85]=97    ;
2212:  !R[86] "INF_PICK_OFFSET" 50mm/sec ;
2213:  R[86]=0    ;
2214:  !R[87] "MAIN_LOAD_OFFSET" (PRELOA ;
2215:  R[87]=100    ;
2216:  !R[100] "GRIPPER_ID" 3 values ;
2217:  !If =100, ID Grippers Installed ;
2218:  !If =200, OD Grippers Installed ;
2219:  !If =300, OD 45 Degree Grippers ;
2220:  R[100]=200    ;
2221:  !--------------------------- ;
2222:   ;
2223:  !If using previous setup data ;
2224:  IF (R[71]=7436) THEN ;
2225:   ;
2226:  !--------------------------- ;
2227:  !1st: Height of Raw piece ;
2228:  R[190]=40.94    ;
2229:  !2nd: Height of Finish piece ;
2230:  R[191]=34.36    ;
2231:  !3rd: Infeed Height Offset ;
2232:  R[192]=55    ;
2233:  !4th: Outfeed Height Offset ;
2234:  R[193]=90    ;
2235:  !--------------------------- ;
2236:   ;
2237:  CALL CREATE_REG(R[190],R[191],R[192],R[193]) ;
2238:   ;
2239:  ENDIF ;
2240:   ;
2241:  !If new loading or offloading pos ;
2242:  !SET R[104] "IMPORT_LOADPOS" ;
2243:  !SET R[104]=1000, Otherwise NO ;
2244:  R[104]=1000    ;
2245:  IF (R[104]=1000) THEN ;
2246:  !R[260]=43, Preload Pos1 ;
2247:  !R[270]=44, Preload PosFinal ;
2248:  !R[300]=53, Offload PosFinal ;
2249:  !PR[43] Pre-Loading Pos1 ;
2250:  CALL CREATE_PR(43,165.493,(-63.481),205.919,144.694,89.018,142.632) ;
2251:  !PR[44] Final Loading Position ;
2252:  CALL CREATE_PR(44,165.659,(-63.704),217.502,144.757,89.017,142.689) ;
2253:  !PR[53] Pre Unloading Position ;
2254:  CALL CREATE_PR(53,(-133.411),92.581,310.76,(-156.985),(-87.994),158.783) ;
2255:  !PR[54] Final Unloading Position ;
2256:  CALL CREATE_PR(54,(-132.12),92.181,271.415,(-156.996),(-87.997),158.789) ;
2257:  !PR[56] assitant Unloading preses ;
2258:  CALL CREATE_PR(56,(-135.297),92.538,351.803,(-156.279),(-87.981),158.047) ;
2259:  !PR[57] assitant Unloading preses ;
2260:  CALL CREATE_PR(57,(-136.348),92.89,384.48,(-156.272),(-87.98),158.048) ;
2261:  !PR[58] assitant Unloading preses ;
2262:  CALL CREATE_PR(58,(-136.985),93.066,404.648,(-156.269),(-87.977),158.046) ;
2263:  ENDIF ;
2264:   ;
2265:  !---------------------------- ;
2266:  !SR[2] = "JOB_VAR_OD_GRIP" ;
2267:  !JOB_VAR_COMMON(R[103])'s value ;
2268:  !---------------------------- ;
2269:  !2By3 SR[2] INF, Max 18(Straight) ;
2270:  !R[103]=200 ;
2271:  !2By3 INF 45 Degree Diagonal Shif ;
2272:  !R[103]=210 ;
2273:  !---------------------------- ;
2274:  !3By4 SR[2] INF, Max 36(Straight) ;
2275:  !R[103]=250 ;
2276:  !3By4 INF 45 Degree Diagonal Shif ;
2277:  !R[103]=260 ;
2278:  !---------------------------- ;
2279:  !R[103] "JOB_PROFILE" Selection ;
2280:  R[103]=270    ;
2281:  CALL JOB_VAR_COMMON(R[103]) ;
2282:   ;
2283:  ENDIF ;
2284:   ;
2285:  JMP LBL[9999] ;
2286:   ;
2287:  !Job 102577436 Logic Ends ;
2288:  !--------------------------- ;
2289:   ;
2290:  LBL[7688] ;
2291:  !--------------------------- ;
2292:  !PORT-DRAIN PAL ;
2293:  !Item 1017688 , Rev A ;
2294:  !Last Modified: 2025-03-25 ;
2295:  !Modified by: Aaron ;
2296:  !0.625 IN Height ;
2297:  !1.202 IN ID, 2.25 IN OD ;
2298:  !OD Jaw # 2009 ;
2299:  !------------------------- ;
2300:  IF (R[70]=7688) THEN ;
2301:   ;
2302:  !Define Parameters for INF/OTF ;
2303:  !R[105]=AR[1]=100, 2By3 Sheet ;
2304:  !R[105]=AR[1]=200, 3By4 Sheet ;
2305:  !R[105]=AR[1]=300, 5By7 Sheet ;
2306:  CALL JOB_VAR_SETUP(400) ;
2307:   ;
2308:  !------------------------- ;
2309:  !Define Parameters for Job ;
2310:  R[1]=1    ;
2311:  R[67]=25    ;
2312:  R[2]=0    ;
2313:  R[139]=12    ;
2314:  R[3]=0    ;
2315:  R[4]=0    ;
2316:  R[85]=65    ;
2317:  R[86]=0    ;
2318:  R[87]=150    ;
2319:  R[95]=100    ;
2320:  R[110]=2026    ;
2321:  !CNC W-AXIS OFFSET ;
2322:  R[111]=((-16.06)) ;
2323:  !X-Compliance Push Bypass ;
2324:  F[6:OFF]=(OFF) ;
2325:  !--------------------------- ;
2326:  !R[100] "GRIPPER_ID" 3 values ;
2327:  !If =100, ID Grippers Installed ;
2328:  !If =200, OD Grippers Installed ;
2329:  !If =300, OD 45 Degree Grippers ;
2330:  R[100]=200    ;
2331:  !--------------------------- ;
2332:   ;
2333:  !If using previous setup data ;
2334:  IF (R[71]=7688) THEN ;
2335:   ;
2336:  !--------------------------- ;
2337:  R[190]=20.5    ;
2338:  R[191]=15.798    ;
2339:  R[192]=(-45)    ;
2340:  R[193]=(-55)    ;
2341:  !--------------------------- ;
2342:   ;
2343:   ;
2344:  CALL CREATE_REG(R[190],R[191],R[192],R[193]) ;
2345:   ;
2346:  ENDIF ;
2347:   ;
2348:  !If new loading or offloading pos ;
2349:  !SET R[104] "IMPORT_LOADPOS" ;
2350:  !SET R[104]=1000, Otherwise NO ;
2351:  R[104]=1000    ;
2352:  IF (R[104]=1000) THEN ;
2353:  !R[260]=43, Preload Pos1 ;
2354:  !R[270]=44, Preload PosFinal ;
2355:  !R[300]=53, Offload PosFinal ;
2356:  !PR[43] Pre-Loading Pos1 ;
2357:  CALL CREATE_PR(43,166.287,(-60.554),326.39,167.368,88.183,166.842) ;
2358:  !PR[44] Final Loading Position ;
2359:  CALL CREATE_PR(44,166.634,(-60.5),336.871,167.345,88.177,166.825) ;
2360:  !PR[53] Pre Unloading Position ;
2361:  CALL CREATE_PR(53,(-125.562),94.788,24.296,160.83,(-88.401),(-160.179)) ;
2362:  !PR[54] Final Unloading Position ;
2363:  CALL CREATE_PR(54,(-124.782),94.781,(-4.113),160.935,(-88.4),(-160.272)) ;
2364:  ENDIF ;
2365:   ;
2366:  !---------------------------- ;
2367:  !SR[2] = "JOB_VAR_OD_GRIP" ;
2368:  !JOB_VAR_COMMON(R[103])'s value ;
2369:  !---------------------------- ;
2370:  !2By3 SR[2] INF, Max 18(Straight) ;
2371:  !R[103]=200 ;
2372:  !2By3 INF 45 Degree Diagonal Shif ;
2373:  !R[103]=210 ;
2374:  !---------------------------- ;
2375:  !3By4 SR[2] INF, Max 36(Straight) ;
2376:  !R[103]=250 ;
2377:  !3By4 INF 45 Degree Diagonal Shif ;
2378:  !R[103]=260 ;
2379:  !---------------------------- ;
2380:  !R[103] "JOB_PROFILE" Selection ;
2381:  R[103]=280    ;
2382:  CALL JOB_VAR_COMMON(R[103]) ;
2383:   ;
2384:  ENDIF ;
2385:   ;
2386:  JMP LBL[9999] ;
2387:   ;
2388:  !Job 1017688 Logic Ends ;
2389:  !--------------------------- ;
2390:   ;
2391:  LBL[7757] ;
2392:  !--------------------------- ;
2393:  !RAYTHEON, TUMBLER ;
2394:  !Item 207757 , Rev A ;
2395:  !Last Modified: 2025-04-23 ;
2396:  !Modified by: Aaron ;
2397:  !0.625 IN Height ;
2398:  !1.202 IN ID, 2.25 IN OD ;
2399:  !OD Jaw # 2012 ;
2400:  !------------------------- ;
2401:  IF (R[70]=7757) THEN ;
2402:   ;
2403:  !Define Parameters for INF/OTF ;
2404:  !R[105]=AR[1]=100, 2By3 Sheet ;
2405:  !R[105]=AR[1]=200, 3By4 Sheet ;
2406:  !R[105]=AR[1]=300, 5By7 Sheet ;
2407:  CALL JOB_VAR_SETUP(220) ;
2408:   ;
2409:  !------------------------- ;
2410:  !Define Parameters for Job ;
2411:  R[1]=1    ;
2412:  R[67]=20    ;
2413:  R[2]=0    ;
2414:  R[139]=12    ;
2415:  R[3]=0    ;
2416:  R[4]=0    ;
2417:  R[85]=64    ;
2418:  R[86]=0    ;
2419:  R[87]=150    ;
2420:  R[95]=100    ;
2421:  R[110]=2026    ;
2422:  !CNC W-AXIS OFFSET ;
2423:  R[111]=((-16.06)) ;
2424:  !X-Compliance Push Bypass ;
2425:  F[6:OFF]=(OFF) ;
2426:  !--------------------------- ;
2427:  !R[100] "GRIPPER_ID" 3 values ;
2428:  !If =100, ID Grippers Installed ;
2429:  !If =200, OD Grippers Installed ;
2430:  !If =300, OD 45 Degree Grippers ;
2431:  R[100]=200    ;
2432:  !--------------------------- ;
2433:   ;
2434:  !If using previous setup data ;
2435:  IF (R[71]=7757) THEN ;
2436:   ;
2437:  !--------------------------- ;
2438:  R[190]=47.13    ;
2439:  R[191]=15.798    ;
2440:  R[192]=369    ;
2441:  R[193]=(-498)    ;
2442:  !--------------------------- ;
2443:   ;
2444:   ;
2445:  CALL CREATE_REG(R[190],R[191],R[192],R[193]) ;
2446:   ;
2447:  ENDIF ;
2448:   ;
2449:  !If new loading or offloading pos ;
2450:  !SET R[104] "IMPORT_LOADPOS" ;
2451:  !SET R[104]=1000, Otherwise NO ;
2452:  R[104]=1000    ;
2453:  IF (R[104]=1000) THEN ;
2454:  !R[260]=43, Preload Pos1 ;
2455:  !R[270]=44, Preload PosFinal ;
2456:  !R[300]=53, Offload PosFinal ;
2457:  !PR[43] Pre-Loading Pos1 ;
2458:  CALL CREATE_PR(43,165.481,(-61.288),311.872,(-174.717),88.15,(-176.825)) ;
2459:  !PR[44] Final Loading Position ;
2460:  CALL CREATE_PR(44,166.248,(-60.915),335.121,(-174.8),88.142,(-176.894)) ;
2461:  !PR[53] Pre Unloading Position ;
2462:  CALL CREATE_PR(53,(-127.197),94.302,111.215,163.187,(-88.443),(-162.218)) ;
2463:  !PR[54] Final Unloading Position ;
2464:  CALL CREATE_PR(54,(-124.097),94.652,(-5.746),163.578,(-88.445),(-162.58)) ;
2465:  ENDIF ;
2466:   ;
2467:  !---------------------------- ;
2468:  !SR[2] = "JOB_VAR_OD_GRIP" ;
2469:  !JOB_VAR_COMMON(R[103])'s value ;
2470:  !---------------------------- ;
2471:  !2By3 SR[2] INF, Max 18(Straight) ;
2472:  !R[103]=200 ;
2473:  !2By3 INF 45 Degree Diagonal Shif ;
2474:  !R[103]=210 ;
2475:  !---------------------------- ;
2476:  !3By4 SR[2] INF, Max 36(Straight) ;
2477:  !R[103]=250 ;
2478:  !3By4 INF 45 Degree Diagonal Shif ;
2479:  !R[103]=260 ;
2480:  !---------------------------- ;
2481:  !R[103] "JOB_PROFILE" Selection ;
2482:  R[103]=340    ;
2483:  CALL JOB_VAR_COMMON(R[103]) ;
2484:   ;
2485:  ENDIF ;
2486:   ;
2487:  JMP LBL[9999] ;
2488:   ;
2489:  !Job 207757 Logic Ends ;
2490:  !--------------------------- ;
2491:   ;
2492:  LBL[8034] ;
2493:  !--------------------------- ;
2494:  !Housing Motor ;
2495:  !Item 198034 , Rev B ;
2496:  !Last Modified: 2025-07-30 ;
2497:  !Modified by: Aaron ;
2498:  !2.68 IN Height ;
2499:  !1.8 IN ID,3.111 OD ;
2500:  !OD Jaw # 2007 ;
2501:  !--------------------------- ;
2502:  IF (R[70]=8034) THEN ;
2503:   ;
2504:  !Define Parameters for INF/OTF ;
2505:  !R[105]=AR[1]=100, 2By3 Sheet ;
2506:  !R[105]=AR[1]=200, 3By4 Sheet ;
2507:  !R[105]=AR[1]=300, 5By7 Sheet ;
2508:  CALL JOB_VAR_SETUP(100) ;
2509:   ;
2510:  !------------------------- ;
2511:  !Define Parameters for Job ;
2512:  R[1]=1    ;
2513:  R[67]=20    ;
2514:  R[2]=0    ;
2515:  R[139]=12    ;
2516:  R[3]=0    ;
2517:  R[4]=0    ;
2518:  R[85]=64    ;
2519:  R[86]=0    ;
2520:  R[87]=150    ;
2521:  R[95]=100    ;
2522:  R[110]=2026    ;
2523:  !CNC W-AXIS OFFSET ;
2524:  R[111]=((-14.17)) ;
2525:  !X-Compliance Push Bypass ;
2526:  F[6:OFF]=(OFF) ;
2527:  !--------------------------- ;
2528:  !R[100] "GRIPPER_ID" 3 values ;
2529:  !If =100, ID Grippers Installed ;
2530:  !If =200, OD Grippers Installed ;
2531:  !If =300, OD 45 Degree Grippers ;
2532:  R[100]=200    ;
2533:  !--------------------------- ;
2534:   ;
2535:  !If using previous setup data ;
2536:  IF (R[71]=8034) THEN ;
2537:   ;
2538:  !--------------------------- ;
2539:  R[190]=90.3    ;
2540:  R[191]=71    ;
2541:  R[192]=369    ;
2542:  R[193]=(-498)    ;
2543:  !--------------------------- ;
2544:   ;
2545:   ;
2546:  CALL CREATE_REG(R[190],R[191],R[192],R[193]) ;
2547:   ;
2548:  ENDIF ;
2549:   ;
2550:  !If new loading or offloading pos ;
2551:  !SET R[104] "IMPORT_LOADPOS" ;
2552:  !SET R[104]=1000, Otherwise NO ;
2553:  R[104]=1000    ;
2554:  IF (R[104]=1000) THEN ;
2555:  !R[260]=43, Preload Pos1 ;
2556:  !R[270]=44, Preload PosFinal ;
2557:  !R[300]=53, Offload PosFinal ;
2558:  !PR[43] Pre-Loading Pos1 ;
2559:  CALL CREATE_PR(43,165.481,(-61.288),311.872,(-174.717),88.15,(-176.825)) ;
2560:  !PR[44] Final Loading Position ;
2561:  CALL CREATE_PR(44,166.248,(-60.915),335.121,(-174.8),88.142,(-176.894)) ;
2562:  !PR[53] Pre Unloading Position ;
2563:  CALL CREATE_PR(53,(-127.197),94.302,111.215,163.187,(-88.443),(-162.218)) ;
2564:  !PR[54] Final Unloading Position ;
2565:  CALL CREATE_PR(54,(-124.097),94.652,(-5.746),163.578,(-88.445),(-162.58)) ;
2566:  ENDIF ;
2567:   ;
2568:  !---------------------------- ;
2569:  !SR[2] = "JOB_VAR_OD_GRIP" ;
2570:  !JOB_VAR_COMMON(R[103])'s value ;
2571:  !---------------------------- ;
2572:  !2By3 SR[2] INF, Max 18(Straight) ;
2573:  !R[103]=200 ;
2574:  !2By3 INF 45 Degree Diagonal Shif ;
2575:  !R[103]=210 ;
2576:  !---------------------------- ;
2577:  !3By4 SR[2] INF, Max 36(Straight) ;
2578:  !R[103]=250 ;
2579:  !3By4 INF 45 Degree Diagonal Shif ;
2580:  !R[103]=260 ;
2581:  !---------------------------- ;
2582:  !R[103] "JOB_PROFILE" Selection ;
2583:  R[103]=200    ;
2584:  CALL JOB_VAR_COMMON(R[103]) ;
2585:   ;
2586:  ENDIF ;
2587:   ;
2588:  JMP LBL[9999] ;
2589:   ;
2590:  !Job 207757 Logic Ends ;
2591:  !--------------------------- ;
2592:  LBL[8902] ;
2593:  !--------------------------- ;
2594:  !Retainer Lower ;
2595:  !Item 102678902 , Rev A ;
2596:  !Last Modified: 2024-07-04 ;
2597:  !Modified by: SH ;
2598:  !1.83 IN Height ;
2599:  !3.6 IN ID, 4.5 IN OD ;
2600:  !OD Jaw # 2003 ;
2601:  !--------------------------- ;
2602:  IF (R[70]=8902) THEN ;
2603:  !Define Parameters for INF/OTF ;
2604:  !R[105]=AR[1]=100, 2By3 Sheet ;
2605:  !R[105]=AR[1]=200, 3By4 Sheet ;
2606:  !R[105]=AR[1]=300, 5By7 Sheet ;
2607:  CALL JOB_VAR_SETUP(100) ;
2608:   ;
2609:  !--------------------------- ;
2610:  !Define Parameters for Job ;
2611:  R[1]=1    ;
2612:  R[67]=20    ;
2613:  R[2]=0    ;
2614:  R[139]=5    ;
2615:  !R[85] "INF_JAW_OFFSET"(Hgt) ;
2616:  R[85]=30    ;
2617:  !R[86] "INF_PICK_OFFSET" 50mm/sec ;
2618:  R[86]=5    ;
2619:  !R[87] "MAIN_LOAD_OFFSET" (PRELOA ;
2620:  R[87]=100    ;
2621:  !R[100] "GRIPPER_ID" 3 values ;
2622:  !If =100, ID Grippers Installed ;
2623:  !If =200, OD Grippers Installed ;
2624:  !If =300, OD 45 Degree Grippers ;
2625:  R[100]=200    ;
2626:  !--------------------------- ;
2627:   ;
2628:  !If using previous setup data ;
2629:  IF (R[71]=8902) THEN ;
2630:   ;
2631:  !--------------------------- ;
2632:  !1st: Height of Raw piece ;
2633:  R[190]=1.5    ;
2634:  !2nd: Height of Finish piece ;
2635:  R[191]=1.06    ;
2636:  !3rd: Infeed Height Offset ;
2637:  R[192]=(-213)    ;
2638:  !4th: Outfeed Height Offset ;
2639:  R[193]=(-290)    ;
2640:  !--------------------------- ;
2641:   ;
2642:  CALL CREATE_REG(R[190],R[191],R[192],R[193]) ;
2643:   ;
2644:  ENDIF ;
2645:   ;
2646:  !If new loading or offloading pos ;
2647:  !SET R[104] "IMPORT_LOADPOS" ;
2648:  !SET R[104]=1000, Otherwise NO ;
2649:  R[104]=1000    ;
2650:  IF (R[104]=1000) THEN ;
2651:  !R[260]=43, Preload Pos1 ;
2652:  !R[270]=44, Preload PosFinal ;
2653:  !R[300]=53, Offload PosFinal ;
2654:  !PR[43] Pre-Loading Pos1 ;
2655:  CALL CREATE_PR(43,166.108,(-62.03),320.63,160.717,89.189,158.679) ;
2656:  !PR[44] Final Loading Position ;
2657:  CALL CREATE_PR(44,166.98,(-62.044),342.44,160.75,89.185,158.724) ;
2658:  !PR[53] Pre Unloading Position ;
2659:  CALL CREATE_PR(53,(-128.808),94.74,139.95,168.21,(-88.32),(-169.192)) ;
2660:  !PR[54] Final Unloading Position ;
2661:  CALL CREATE_PR(54,(-128.009),95.025,112.33,168.149,(-88.32),(-169.132)) ;
2662:  !PR[56] assitant Unloading preses ;
2663:  CALL CREATE_PR(56,(-131.536),105.713,233.177,173.746,(-88.233),(-175.647)) ;
2664:  !PR[57] assitant Unloading preses ;
2665:  CALL CREATE_PR(57,(-133.703),92.431,364.782,167.802,(-88.383),(-166.755)) ;
2666:  !PR[58] assitant Unloading preses ;
2667:  CALL CREATE_PR(58,(-133.703),92.431,364.782,167.804,(-88.383),(-166.755)) ;
2668:  ENDIF ;
2669:   ;
2670:  !---------------------------- ;
2671:  !SR[2] = "JOB_VAR_OD_GRIP" ;
2672:  !JOB_VAR_COMMON(R[103])'s value ;
2673:  !---------------------------- ;
2674:  !2By3 SR[2] INF, Max 18(Straight) ;
2675:  !R[103]=200 ;
2676:  !2By3 INF 45 Degree Diagonal Shif ;
2677:  !R[103]=210 ;
2678:  !---------------------------- ;
2679:  !3By4 SR[2] INF, Max 36(Straight) ;
2680:  !R[103]=250 ;
2681:  !3By4 INF 45 Degree Diagonal Shif ;
2682:  !R[103]=260 ;
2683:  !---------------------------- ;
2684:  !R[103] "JOB_PROFILE" Selection ;
2685:  R[103]=200    ;
2686:  CALL JOB_VAR_COMMON(R[103]) ;
2687:   ;
2688:  ENDIF ;
2689:   ;
2690:  JMP LBL[9999] ;
2691:   ;
2692:  !Job 102678902 Logic Ends ;
2693:  !--------------------------- ;
2694:   ;
2695:  LBL[9487] ;
2696:  !--------------------------- ;
2697:  !Sub Top ;
2698:  !Item 102709487 , Rev A ;
2699:  !Last Modified: 2024-06-24 ;
2700:  !Modified by: Tsuu ;
2701:  !6.00 IN Height ;
2702:  !2.281 IN ID, 3.25 ;
2703:  !OD Jaw #2010 ;
2704:  !--------------------------- ;
2705:  IF (R[70]=9487) THEN ;
2706:  !Define Parameters for INF/OTF ;
2707:  !R[105]=AR[1]=100, 2By3 Sheet ;
2708:  !R[105]=AR[1]=200, 3By4 Sheet ;
2709:  !R[105]=AR[1]=210, 3By4 Sheet Man ;
2710:  !R[105]=AR[1]=300, 5By7 Sheet ;
2711:  CALL JOB_VAR_SETUP(200) ;
2712:   ;
2713:  !--------------------------- ;
2714:  !Define Parameters for Job ;
2715:  R[1]=1    ;
2716:  R[67]=25    ;
2717:  R[2]=1    ;
2718:  R[139]=22    ;
2719:  !R[85] "INF_JAW_OFFSET"(Hgt) ;
2720:  R[85]=35    ;
2721:  !R[86] "INF_PICK_OFFSET" 50mm/sec ;
2722:  R[86]=25    ;
2723:  !R[87] "MAIN_LOAD_OFFSET" (PRELOA ;
2724:  R[87]=0    ;
2725:  !R[100] "GRIPPER_ID" 3 values ;
2726:  !If =100, ID Grippers Installed ;
2727:  !If =200, OD Grippers Installed ;
2728:  !If =300, OD 45 Degree Grippers ;
2729:  R[100]=200    ;
2730:  !--------------------------- ;
2731:   ;
2732:  !If using previous setup data ;
2733:  IF (R[71]=9487) THEN ;
2734:   ;
2735:  !--------------------------- ;
2736:  !1st: Height of Raw piece ;
2737:  R[190]=157.48    ;
2738:  !2nd: Height of Finish piece ;
2739:  R[191]=152.399    ;
2740:  !3rd: Infeed Height Offset ;
2741:  R[192]=(-72)    ;
2742:  !4th: Outfeed Height Offset ;
2743:  R[193]=(-390)    ;
2744:  !--------------------------- ;
2745:   ;
2746:  CALL CREATE_REG(R[190],R[191],R[192],R[193]) ;
2747:   ;
2748:  ENDIF ;
2749:   ;
2750:  !If new loading or offloading pos ;
2751:  !SET R[104] "IMPORT_LOADPOS" ;
2752:  !SET R[104]=1000, Otherwise NO ;
2753:  R[104]=1000    ;
2754:  IF (R[104]=1000) THEN ;
2755:  !R[260]=43, Preload Pos1 ;
2756:  !R[270]=44, Preload PosFinal ;
2757:  !R[300]=53, Offload PosFinal ;
2758:  !PR[43] Pre-Loading Pos1 ;
2759:  CALL CREATE_PR(43,166.27,(-59.94),245.259,135.47,88.65,133.399) ;
2760:  !PR[44] Final Loading Position ;
2761:  CALL CREATE_PR(44,168.05,(-60.983),277.622,135.319,88.673,133.228) ;
2762:  !PR[53] Pre Unloading Position ;
2763:  CALL CREATE_PR(53,(-132.097),93.918,201.582,171.779,(-88.303),(-173.664)) ;
2764:  !PR[54] Final Unloading Position ;
2765:  CALL CREATE_PR(54,(-129.876),94.29,125.692,171.712,(-88.304),(-173.603)) ;
2766:  !PR[56] assitant Unloading preses ;
2767:  CALL CREATE_PR(56,(-131.298),94.552,188.064,173.651,(-88.242),(-175.595)) ;
2768:  !PR[57] assitant Unloading preses ;
2769:  CALL CREATE_PR(57,(-133.938),94.235,274.821,173.733,(-88.241),(-175.673)) ;
2770:  !PR[58] assitant Unloading preses ;
2771:  CALL CREATE_PR(58,(-136.182),93.951,348.894,173.814,(-88.239),(-175.748)) ;
2772:  !PR[59] assitant Unloading preses ;
2773:  CALL CREATE_PR(59,82.383,234.843,398.401,(-92.773),(-50.7),90.238) ;
2774:  ENDIF ;
2775:   ;
2776:  !---------------------------- ;
2777:  !SR[2] = "JOB_VAR_OD_GRIP" ;
2778:  !JOB_VAR_COMMON(R[103])'s value ;
2779:  !---------------------------- ;
2780:  !2By3 SR[2] INF, Max 18(Straight) ;
2781:  !R[103]=200 ;
2782:  !2By3 INF 45 Degree Diagonal Shif ;
2783:  !R[103]=210 ;
2784:  !---------------------------- ;
2785:  !3By4 SR[2] INF, Max 36(Straight) ;
2786:  !R[103]=250 ;
2787:  !3By4 INF Mandrel, 2 Trays ;
2788:  !R[103]=260 ;
2789:  !---------------------------- ;
2790:  !R[103] "JOB_PROFILE" Selection ;
2791:  R[103]=250    ;
2792:  CALL JOB_VAR_COMMON(R[103]) ;
2793:   ;
2794:  ENDIF ;
2795:   ;
2796:  JMP LBL[9999] ;
2797:   ;
2798:  !Job 102709487 Logic Ends ;
2799:  !--------------------------- ;
2800:   ;
2801:  LBL[9654] ;
2802:  !--------------------------- ;
2803:  !ADPTR ;
2804:  !Item 100009654, Rev B ;
2805:  !Last Modified: 2026-04-02 ;
2806:  !Modified by: Aaron ;
2807:  !6.25 IN Height ;
2808:  !3.16 IN ID, 3.742 IN OD 25.5 Lbs ;
2809:  !OD Jaw #2004 ;
2810:  !------------------------- ;
2811:  IF (R[70]=9654) THEN ;
2812:   ;
2813:  !Define Parameters for INF/OTF ;
2814:  !R[105]=AR[1]=100, 2By3 Sheet ;
2815:  !R[105]=AR[1]=200, 3By4 Sheet ;
2816:  !R[105]=AR[1]=300, 5By7 Sheet ;
2817:  CALL JOB_VAR_SETUP(100) ;
2818:   ;
2819:  !------------------------- ;
2820:  !Define Parameters for Job ;
2821:  R[1]=1    ;
2822:  R[67]=30    ;
2823:  R[2]=1    ;
2824:  R[139]=12    ;
2825:  R[3]=0    ;
2826:  R[4]=0    ;
2827:  R[85]=116.22    ;
2828:  R[86]=5    ;
2829:  R[87]=150    ;
2830:  R[95]=100    ;
2831:  R[110]=2004    ;
2832:  !CNC W-AXIS OFFSET ;
2833:  R[111]=((-16.06)) ;
2834:  !X-Compliance Push Bypass ;
2835:  F[6:OFF]=(OFF) ;
2836:  !--------------------------- ;
2837:  !R[100] "GRIPPER_ID" 3 values ;
2838:  !If =100, ID Grippers Installed ;
2839:  !If =200, OD Grippers Installed ;
2840:  !If =300, OD 45 Degree Grippers ;
2841:  R[100]=200    ;
2842:  !--------------------------- ;
2843:   ;
2844:  !If using previous setup data ;
2845:  IF (R[71]=9654) THEN ;
2846:   ;
2847:  !--------------------------- ;
2848:  R[190]=159.28    ;
2849:  R[191]=158.75    ;
2850:  R[192]=(-317)    ;
2851:  R[193]=(-225)    ;
2852:  !--------------------------- ;
2853:   ;
2854:   ;
2855:  CALL CREATE_REG(R[190],R[191],R[192],R[193]) ;
2856:   ;
2857:  ENDIF ;
2858:   ;
2859:  !If new loading or offloading pos ;
2860:  !SET R[104] "IMPORT_LOADPOS" ;
2861:  !SET R[104]=1000, Otherwise NO ;
2862:  R[104]=1000    ;
2863:  IF (R[104]=1000) THEN ;
2864:  !R[260]=43, Preload Pos1 ;
2865:  !R[270]=44, Preload PosFinal ;
2866:  !R[300]=53, Offload PosFinal ;
2867:  !PR[43] Pre-Loading Pos1 ;
2868:  CALL CREATE_PR(43,160.369,(-64.368),163.94,178.858,88.075,176.797) ;
2869:  !PR[44] Final Loading Position ;
2870:  CALL CREATE_PR(44,165.32,(-64.498),311.312,178.955,88.074,176.901) ;
2871:  !PR[53] Pre Unloading Position ;
2872:  CALL CREATE_PR(53,(-128.207),92.924,159.495,160.343,(-88.417),(-159.311)) ;
2873:  !PR[54] Final Unloading Position ;
2874:  CALL CREATE_PR(54,(-124.447),94.192,14.339,160.537,(-88.418),(-159.498)) ;
2875:  ENDIF ;
2876:   ;
2877:  !---------------------------- ;
2878:  !SR[2] = "JOB_VAR_OD_GRIP" ;
2879:  !JOB_VAR_COMMON(R[103])'s value ;
2880:  !---------------------------- ;
2881:  !2By3 SR[2] INF, Max 18(Straight) ;
2882:  !R[103]=200 ;
2883:  !2By3 INF 45 Degree Diagonal Shif ;
2884:  !R[103]=210 ;
2885:  !---------------------------- ;
2886:  !3By4 SR[2] INF, Max 36(Straight) ;
2887:  !R[103]=250 ;
2888:  !3By4 INF 45 Degree Diagonal Shif ;
2889:  !R[103]=260 ;
2890:  !---------------------------- ;
2891:  !R[103] "JOB_PROFILE" Selection ;
2892:  R[103]=200    ;
2893:  CALL JOB_VAR_COMMON(R[103]) ;
2894:   ;
2895:  ENDIF ;
2896:   ;
2897:  JMP LBL[9999] ;
2898:   ;
2899:  !Job 100009654 Logic Ends ;
2900:  !--------------------------- ;
2901:   ;
2902:  LBL[9700] ;
2903:  !--------------------------- ;
2904:  !Ring,Spacer ;
2905:  !Item 102779700 , Rev B ;
2906:  !Last Modified: 2022-10-06 ;
2907:  !Modified by: Tsuu ;
2908:  !0.75 IN Height ;
2909:  !1.610 IN ID, 3.20 IN OD ;
2910:  !ID Jaw # 2007 ;
2911:  !--------------------------- ;
2912:  IF (R[70]=9700) THEN ;
2913:  !Define Parameters for INF/OTF ;
2914:  !R[105]=AR[1]=100, 2By3 Sheet ;
2915:  !R[105]=AR[1]=200, 3By4 Sheet ;
2916:  !R[105]=AR[1]=300, 5By7 Sheet ;
2917:  CALL JOB_VAR_SETUP(100) ;
2918:   ;
2919:  !--------------------------- ;
2920:  !Define Parameters for Job ;
2921:  !R[85] "INF_JAW_OFFSET"(Hgt) ;
2922:  R[85]=200    ;
2923:  !R[86] "INF_PICK_OFFSET" 50mm/sec ;
2924:  R[86]=2    ;
2925:  !R[87] "MAIN_LOAD_OFFSET" (PRELOA ;
2926:  R[87]=100    ;
2927:  !R[100] "GRIPPER_ID" 3 values ;
2928:  !If =100, ID Grippers Installed ;
2929:  !If =200, OD Grippers Installed ;
2930:  !If =300, OD 45 Degree Grippers ;
2931:  R[100]=200    ;
2932:  !--------------------------- ;
2933:   ;
2934:  !If using previous setup data ;
2935:  IF (R[71]=9700) THEN ;
2936:   ;
2937:  !--------------------------- ;
2938:  !1st: Height of Raw piece ;
2939:  R[190]=21.84    ;
2940:  !2nd: Height of Finish piece ;
2941:  R[191]=19.05    ;
2942:  !3rd: Infeed Height Offset ;
2943:  R[192]=(-140)    ;
2944:  !4th: Outfeed Height Offset ;
2945:  R[193]=(-202)    ;
2946:  !--------------------------- ;
2947:   ;
2948:  CALL CREATE_REG(R[190],R[191],R[192],R[193]) ;
2949:   ;
2950:  ENDIF ;
2951:   ;
2952:  !If new loading or offloading pos ;
2953:  !SET R[104] "IMPORT_LOADPOS" ;
2954:  !SET R[104]=1000, Otherwise NO ;
2955:  R[104]=1000    ;
2956:  IF (R[104]=1000) THEN ;
2957:  !R[260]=43, Preload Pos1 ;
2958:  !R[270]=44, Preload PosFinal ;
2959:  !R[300]=53, Offload PosFinal ;
2960:  !PR[43] Pre-Loading Pos1 ;
2961:  CALL CREATE_PR(43,164.613,(-61.339),204.384,160.683,89.19,158.634) ;
2962:  !PR[44] Final Loading Position ;
2963:  CALL CREATE_PR(44,164.819,(-61.517),218.821,160.664,89.188,158.61) ;
2964:  !PR[53] Pre Unloading Position ;
2965:  CALL CREATE_PR(53,(-133.746),93.958,312.88,168.05,(-88.326),(-169.036)) ;
2966:  !PR[54] Final Unloading Position ;
2967:  CALL CREATE_PR(54,(-133.228),94.437,293.638,167.785,(-88.327),(-168.787)) ;
2968:  !PR[56] assitant Unloading preses ;
2969:  CALL CREATE_PR(56,(-131.536),105.713,233.177,173.746,(-88.233),(-175.647)) ;
